_stAxis.stconfig.fReadAxisParameter := fbReadParameter.Value;
mParameters_ReadParameter.Busy := fbReadParameter.Busy;
mParameters_ReadParameter.Done := fbReadParameter.Valid;
mParameters_ReadParameter.Error := fbReadParameter.Error;
mParameters_ReadParameter.ErrorID := fbReadParameter.ErrorID;

IF fbReadParameter.Error THEN
    _stAxis.stError.fbReadParameterErrorId := fbReadParameter.ErrorID;
END_IF
END_METHOD

METHOD mParameters_WriteParameter : ST_McStatus

IF _stAxis.stControl.eCommand = E_MotionFunctions.eWriteParameter THEN
    fbWriteParameter.Execute := _stAxis.stControl.bExecute;
END_IF

fbWriteParameter.ParameterNumber := _stAxis.stConfig.eAxisParameters;
fbWriteParameter.Value := _stAxis.stConfig.fWriteAxisParameter;

fbWriteParameter(Axis := _stAxis.Axis);
fbWriteParameter.Execute := FALSE;

mParameters_WriteParameter.Busy := fbWriteParameter.Busy;
mParameters_WriteParameter.Done := fbWriteParameter.Done;
mParameters_WriteParameter.Error := fbWriteParameter.Error;
mParameters_WriteParameter.ErrorID := fbWriteParameter.ErrorID;

IF fbWriteParameter.Error THEN
    _stAxis.stError.fbWriteParameterErrorId := fbWriteParameter.ErrorID;
END_IF
END_METHOD

METHOD mParameters_WriteSWLimits : ST_McStatus
IF _stAxis.stControl.eCommand = E_MotionFunctions.eWriteToggleSWLimits THEN
    fbWriteSWLimitMax.Execute := _stAxis.stControl.bExecute;
	fbWriteSWLimitMin.Execute := _stAxis.stControl.bExecute;
END_IF

fbWriteSWLimitMax.ParameterNumber := E_AxisParameters.EnableLimitForward;
fbWriteSWLimitMax.Value := _stAxis.stConfig.fWriteAxisBoolParameter;
fbWriteSWLimitMin.ParameterNumber := E_AxisParameters.EnableLimitBackward;
fbWriteSWLimitMin.Value := _stAxis.stConfig.fWriteAxisBoolParameter;

fbWriteSWLimitMax(Axis := _stAxis.Axis);
fbWriteSWLimitMax.Execute := FALSE;
fbWriteSWLimitMin(Axis := _stAxis.Axis);
fbWriteSWLimitMin.Execute := FALSE;

mParameters_WriteSWLimits.Busy := fbWriteSWLimitMax.Busy OR fbWriteSWLimitMin.Busy;
mParameters_WriteSWLimits.Done := fbWriteSWLimitMax.Done OR fbWriteSWLimitMin.Done;
mParameters_WriteSWLimits.Error := fbWriteSWLimitMax.Error OR fbWriteSWLimitMin.Error;
mParameters_WriteSWLimits.ErrorID := fbWriteSWLimitMax.ErrorID OR fbWriteSWLimitMin.ErrorID;

IF fbWriteSWLimitMax.Error OR fbWriteSWLimitMin.Error THEN
    _stAxis.stError.fbWriteParameterErrorId := fbWriteSWLimitMax.ErrorID OR fbWriteSWLimitMin.ErrorID; 
END_IF
END_METHOD

METHOD mStatus_AxisStatus : BOOL

_stAxis.Axis.ReadStatus();
IF _stAxis.Axis.Status.OpMode.Modulo THEN
    _stAxis.stStatus.fActPosition := _stAxis.Axis.NcToPlc.ModuloActPos;
ELSE
    _stAxis.stStatus.fActPosition := _stAxis.Axis.NcToPlc.ActPos;
END_IF

_stAxis.stStatus.bHomed := _stAxis.Axis.Status.Homed;
_stAxis.stStatus.bMoving := _stAxis.Axis.Status.Moving;
_stAxis.stStatus.fActVelocity := _stAxis.Axis.NcToPlc.ActVelo;
_stAxis.stStatus.bMovingForward := _stAxis.Axis.Status.PositiveDirection;
_stAxis.stStatus.bMovingBackward := _stAxis.Axis.Status.NegativeDirection;
_stAxis.stStatus.bInTargetPosition := _stAxis.Axis.Status.InTargetPosition;
//_stAxis.stStatus.bEnabled := _stAxis.Axis.Status.Operational;
_stAxis.stStatus.bEnabled := NOT(_stAxis.Axis.Status.Disabled);	//This is crap but I don't know a better way

_stAxis.stStatus.SPGEnabled := _stAxis.Axis.Status.ExtSetPointGenEnabled;
END_METHOD

METHOD mStatus_Busy : BOOL
VAR
    i: UINT;
    tmpBusy: BOOL;
END_VAR

FOR i := 5 TO 10 DO
    tmpBusy := astMcStatus[i]^.Busy OR tmpBusy;
END_FOR
mStatus_Busy := tmpBusy;
END_METHOD

METHOD mStatus_CommandAborted : BOOL
VAR
    i: UINT;
    tmpCmdAborted: BOOL;
END_VAR

FOR i := 5 TO 9 DO
    tmpCmdAborted := astMcStatus[i]^.CommandAborted OR tmpCmdAborted;
END_FOR

fbCommandAbortedRTrig(CLK := tmpCmdAborted);
IF fbCommandAbortedRTrig.Q THEN
    _stAxis.stStatus.bCommandAborted := TRUE;
END_IF
END_METHOD

METHOD mStatus_Done : BOOL
VAR
    i: UINT;
    tmpDone: BOOL;
END_VAR

FOR i := 5 TO 10 DO
    tmpDone := astMcStatus[i]^.Done OR tmpDone;
END_FOR
//fbDoneRTrig(CLK:= mStatus_Done());
fbDoneRTrig(CLK := tmpDone);
IF fbDoneRTrig.Q THEN
    _stAxis.stStatus.bDone := TRUE;
END_IF
END_METHOD

METHOD mStatus_Error : BOOL
VAR
    i: UINT;
    tmpError: BOOL;

END_VAR

FOR i := 1 TO nMCSTATUS_ARRAY_SIZE DO
    tmpError := astMcStatus[i]^.Error OR tmpError;
END_FOR


fbErrorRTrig(CLK := tmpError);

//Check if NC is in error state and propogate
IF _stAxis.Axis.Status.ErrorStop OR _stAxis.Axis.Status.Error THEN
    _stAxis.stStatus.bError := _stAxis.Axis.Status.ErrorStop OR _stAxis.Axis.Status.Error;
    _stAxis.stStatus.nErrorID := _stAxis.Axis.Status.ErrorID;//NC Error ID
END_IF



IF fbErrorRTrig.Q THEN
        //For each mcStatus
        FOR i := 1 TO nMCSTATUS_ARRAY_SIZE DO
            //If there's an error present propagate
            IF astMcStatus[i]^.ErrorID <> 0 THEN
				_stAxis.stStatus.bMcError := TRUE;
                _stAxis.stStatus.nMcErrorID := astMcStatus[i]^.ErrorID;
            END_IF
        END_FOR
END_IF
END_METHOD

METHOD mStatus_InVelocity : BOOL
VAR
    i: UINT;
    tmpInVelocity: BOOL;
END_VAR
FOR i := 1 TO nMCSTATUS_ARRAY_SIZE DO
    tmpInVelocity := astMcStatus[i]^.InVelocity OR tmpInVelocity;
END_FOR
//fbInVelocityRTrig(CLK:= mStatus_InVelocity());
fbInVelocityRTrig(CLK := tmpInVelocity);
IF fbInVelocityRTrig.Q THEN
    _stAxis.stStatus.bInVelocity := TRUE;
END_IF

fbInVelocityFTrig(CLK := _stAxis.Axis.Status.ContinuousMotion);
IF fbInVelocityFTrig.Q THEN
    _stAxis.stStatus.bInVelocity := FALSE;
END_IF
END_METHOD

METHOD mStatus_Name : BOOL
VAR
	eAxisNames : E_AxisNames;
	sAxisName : STRING;
	sSpace : STRING := ' ';
END_VAR
eAxisNames := TO_INT(GVL.iAxis);
sAxisName := TO_STRING(eAxisNames);
FOR iNameCharacterIndex := 0 TO LEN(sAxisName) DO
	IF  F_ToCHR(sAxisName[iNameCharacterIndex]) = '_' THEN
		sAxisName[iNameCharacterIndex] := sSpace[0];
	END_IF
END_FOR
_stAxis.stDescription.sAxisName := sAxisName;
END_METHOD

METHOD mStatus_NewCommand : BOOL
VAR
    i: UINT;
END_VAR

fbExecuteRTrig(CLK := _stAxis.stControl.bExecute);
IF fbExecuteRTrig.Q THEN
    _stAxis.stStatus.bDone := FALSE;
    _stAxis.stStatus.bCommandAborted := FALSE;

    //On a new motion command, clear the errorID
    CASE _stAxis.stControl.eCommand OF
            E_MotionFunctions.eMoveAbsolute,
            E_MotionFunctions.eMoveRelative,
            E_MotionFunctions.eMoveVelocity,
            E_MotionFunctions.eMoveModulo,
			E_MotionFunctions.eSetPosition,
            E_MotionFunctions.eHome :
                _stAxis.stStatus.nErrorID := 0;
            E_MotionFunctions.eWriteParameter,
            E_MotionFunctions.eReadParameter :
            // Nothing
    END_CASE
END_IF
END_METHOD

METHOD Run : BOOL
mStatus_AxisStatus();
mParameters_ReadNc();
mParameters_Init();
stMcStatusReadParameter := mParameters_ReadParameter();
stMcStatusWriteParameter := mParameters_WriteParameter();
stMcStatusWriteSWLimits := mParameters_WriteSWLimits();

mControl_LimitHitTimer();
mControl_LimitLinking();
mControl_LimitEdge();
stMcStatusPower := mControl_Power();
mControl_AutoEnableDisable();

mControl_EnableSPG();
mControl_DisableSPG();
mControl_FeedSPG();

stMcStatusHalt := mMove_Halt();
stMcStatusStop := mMove_Stop();
stMcStatusReset := mControl_Reset();
stMcStatusSetPosition := mMove_SetPosition();

stMcStatusMoveAbsolute := mMove_MoveAbsolute();
stMcStatusMoveRelative := mMove_MoveRelative();
stMcStatusMoveModulo := mMove_MoveModulo();
stMcStatusMoveVelocity := mMove_MoveVelocity();

stMcStatusLocalMoveAbsolute := mLocalMove_MoveAbsolute();
stMcStatusLocalMoveRelative := mLocalMove_MoveRelative();
stMcStatusLocalMoveVelocity := mLocalMove_MoveVelocity();

stMcStatusHome := mControl_Home();

mStatus_NewCommand();
mStatus_Done();
mStatus_Error();
mStatus_InVelocity();
mStatus_CommandAborted();
_stAxis.stStatus.bBusy := mStatus_Busy();

IF _TaskInfo[fbGetCurTaskIndex.index].FirstCycle THEN
	mStatus_Name();
END_IF


EndOfCycle();
END_METHOD

PROPERTY stAxis : REFERENCE TO ST_AxisStruct
GET
stAxis REF= _stAxis;
END_GET
SET
_stAxis REF= stAxis;
END_SET
END_PROPERTY

END_FUNCTION_BLOCK

// ---- tc_mca_std_lib/POUs/Motion/Homing/FB_Homing.TcPOU
FUNCTION_BLOCK FB_Homing
VAR_IN_OUT
    AxisRef: AXIS_REF;
	
END_VAR
VAR_INPUT
    bExecute: BOOL;
    bLimitFwd: BOOL;
    bLimitBwd: BOOL;
    bHomeSensor: BOOL;
    eHomeSeq: E_HomingRoutines;
    fHomePosition: LREAL;
    fHomeFinishDistance: LREAL;
	fHomeAbsPosition : LREAL;
	bDoAbsoluteMove : BOOL;
	fHomeMidRelativeMove : LREAL;
    stConfig: ST_AxisConfig;
	stHomingConfig : ST_AxisHomingConfig;
	bGoToFwdLimitFirst : BOOL;
	bGoToBwdLimitFirst : BOOL;
	fFastVelocity : LREAL;
END_VAR
VAR_OUTPUT
    bDone : BOOL;
    bBusy: BOOL;
    bCommandAborted: BOOL;
    bError: BOOL;
    nErrorId: UDINT;
	bInHomingSequence: BOOL;
END_VAR
VAR
    //Beckhoff homing function blocks
    fbStepLimitSwitchPreparation: MC_StepLimitSwitchDetection;
    fbStepLimitSwitchDetection: MC_StepLimitSwitchDetection;
    fbStepAbsoluteSwitchDetection: MC_StepAbsoluteSwitchDetection;
	fbStepAbsoluteSwitchPreparation: MC_StepAbsoluteSwitchDetection;
	fbStepReferencePulsePreparation: MC_StepReferencePulseDetection;
    fbStepReferencePulseDetection: MC_StepReferencePulseDetection;
    fbStepBlockLagDetection: MC_StepBlockLagBasedDetection;
    fbHomeDirect: MC_HomeDirect;
    fbSetPos: MC_SetPosition;
    fbFinishHoming: MC_FinishHoming;
    fbAbortHoming: MC_AbortHoming;
	fbMoveRelative : MC_MoveRelative;
	fbMoveAbsolute : MC_MoveAbsolute;
	fbMoveVelocity : MC_MoveVelocity;
    //Hardware Signals
    eLimitSwitchMode: MC_Switch_Mode := mcRisingEdge;
    stLimitSwitchSignal: MC_Ref_Signal_Ref;
    eRefSwitchMode: MC_Switch_Mode := mcRisingEdge;
    stRefSwitchSignal: MC_Ref_Signal_Ref;
    stEncPulseSignal: MC_Ref_Signal_Ref;
    //Homing parameters
    stPreparationDirection: MC_Home_Direction;
    stDetectDirection: MC_Home_Direction;
    stHomingParameter: MC_HomingParameter;
    stOptions: ST_Home_Options4;
    stOptions3: ST_Home_Options3;
    fbVelocityToCam: MC_ReadParameter;
    fVelocityToCam: LREAL;
    fbVelocityFromCam: MC_ReadParameter;
    fVelocityFromCam: LREAL;
    //State machine
    fbExecute: R_TRIG;
    bViaLimitSwitch: BOOL;
	bViaFastEncPulse : BOOL;
	bViaFastRef : BOOL;
    eHomingState: (eWaitForRequest := 0, ePreparation := 1, eDetection := 2, eSetPos := 3, eFinishHoming := 4, eMoveRelative:=5, eAbsMove:=6, eAbortHoming := 20, eGoToFwd:=7, eGoToBwd:=8, eWaitForFwd:=9,eWaitForBwd:=10);
    iErrorId: UDINT;
    bDetectionFB_Execute: BOOL;
    bDetectionFB_Done: BOOL;
    bDetectionFB_Busy: BOOL;
    bDetectionFB_CommandAborted: BOOL;
    bDetectionFB_Error: BOOL;
    nDetectionFB_ErrorID: UDINT;
    fRecordedPosition: LREAL;
    fRecordedPositionLatched: LREAL;
END_VAR

bInHomingSequence:= FALSE;
//Hardware signals
stLimitSwitchSignal.SignalSource := SignalSource_Default;
stLimitSwitchSignal.TouchProbe := PlcEvent;
stRefSwitchSignal.SignalSource := SignalSource_Default;
stRefSwitchSignal.TouchProbe := PlcEvent;
stRefSwitchSignal.Level := bHomeSensor;
stEncPulseSignal.SignalSource := SignalSource_ZeroPulse;
stEncPulseSignal.TouchProbe := TouchProbe1;

fbMoveRelative(
	Axis:= AxisRef, Velocity:= fVelocityToCam);
	fbMoveRelative.Execute:= FALSE;

fbMoveAbsolute(
	Axis:= AxisRef, Velocity:= fFastVelocity, Position:= fHomeAbsPosition);
	fbMoveAbsolute.Execute:= FALSE;

//Constantly read the NC for homing velocities so they are available when a homing is executed
fbVelocityToCam(
    Axis := AxisRef,
    Enable := TRUE,
    ParameterNumber := E_AxisParameters.AxisVelocityToCam,
    ReadMode := READMODE_CYCLIC);

fbVelocityFromCam(
    Axis := AxisRef,
    Enable := TRUE,
    ParameterNumber := E_AxisParameters.AxisVelocityFromCam,
    ReadMode := READMODE_CYCLIC);

    //Only write velocity if the function block has not errored
IF NOT fbVelocityToCam.Error THEN
    fVelocityToCam := fbVelocityToCam.Value;
END_IF

IF NOT fbVelocityFromCam.Error THEN
    fVelocityFromCam := fbVelocityFromCam.Value;
END_IF

    //Feeds function block errors through
IF fbVelocityToCam.Error THEN
    bError := TRUE;
    nErrorID := fbVelocityToCam.ErrorID;

ELSIF fbVelocityFromCam.Error THEN
    bError := TRUE;
    nErrorID := fbVelocityFromCam.ErrorID;
END_IF

//Common function blocks used for all routines
stOptions.DisableDriveAccess := stHomingConfig.bDisableDriveAccess;

//For StepBlockLagDetection
stOptions3.DisableDriveAccess := stHomingConfig.bDisableDriveAccess;

fbStepLimitSwitchPreparation.Options.DisableDriveAccess := stOptions.DisableDriveAccess;
fbStepLimitSwitchPreparation(
    Axis := AxisRef,
    Parameter := stHomingParameter,
    Direction := stPreparationDirection,
    LimitSwitchMode:= eLimitSwitchMode,
    LimitSwitchSignal:= stLimitSwitchSignal,
    Velocity := fVelocityToCam);
	


fbSetPos(
    Axis := AxisRef,
    Position := AxisRef.NcToPlc.ActPos - fRecordedPositionLatched + fHomePosition);

fbFinishHoming.Options.DisableDriveAccess := stOptions.DisableDriveAccess;
fbFinishHoming(
    Axis := AxisRef,
    Parameter := stHomingParameter,
    Velocity := fVelocityFromCam);

fbMoveVelocity(Axis:= AxisRef, Velocity:= ABS(fFastVelocity));
	fbMoveVelocity.Execute:= FALSE;

fbAbortHoming.Options.DisableDriveAccess := stOptions.DisableDriveAccess;
fbAbortHoming(
    Axis := AxisRef,
    Parameter := stHomingParameter);

//ACTs contain function blocks custom to each individual routine for the detection stage
CASE eHomeSeq OF
    E_HomingRoutines.eHomeToLimit_Bwd,
    E_HomingRoutines.eHomeToLimit_Fwd:
        actHomeToLimit();

    E_HomingRoutines.eHomeToRef_Bwd,
	E_HomingRoutines.eHomeToRef_Bwd_Fast,
	E_HomingRoutines.eHomeToRef_Fwd_Fast,
    E_HomingRoutines.eHomeToRef_Fwd:
        actHomeToRef();

    E_HomingRoutines.eHomeToEncPulse_Bwd,
    E_HomingRoutines.eHomeToEncPulse_Fwd,
    E_HomingRoutines.eHomeToEncPulse_viaBwdLimit,
    E_HomingRoutines.eHomeToEncPulse_viaFwdLimit,
	E_HomingRoutines.eHomeToEncPulse_BWD_FAST,
	E_HomingRoutines.eHomeToEncPulse_FWD_FAST:
        actHomeToEncPulse();

    E_HomingRoutines.eHomeToBlock_Bwd,
    E_HomingRoutines.eHomeToBlock_Fwd:
        actHomeToBlock();

    E_HomingRoutines.eHomeDirect:
        actHomeDirect();
END_CASE


//State machine
fbExecute(CLK:= bExecute);
CASE eHomingState OF

    eWaitForRequest:
        IF NOT bExecute THEN
            bBusy := FALSE;
            bDone := FALSE;
            bCommandAborted := FALSE;
            bError := FALSE;
            nErrorID := 0;
            iErrorID := 0;

            fbStepLimitSwitchPreparation.Execute := FALSE;
            fbStepLimitSwitchDetection.Execute := FALSE;
            fbStepAbsoluteSwitchDetection.Execute := FALSE;
			fbStepReferencePulsePreparation.Execute := FALSE;
            fbStepReferencePulseDetection.Execute := FALSE;
            fbStepBlockLagDetection.Execute := FALSE;
            fbHomeDirect.Execute := FALSE;
            fbSetPos.Execute := FALSE;
            fbFinishHoming.Execute := FALSE;
            fbAbortHoming.Execute := FALSE;
        END_IF

        IF fbExecute.Q AND NOT(eHomeSeq = E_HomingRoutines.eNoHoming)THEN
            bBusy:= TRUE;
			IF bGoToFwdLimitFirst THEN
				eHomingState:= eGoToFwd;
			ELSIF bGoToBwdLimitFirst THEN
				eHomingState:= eGoToBwd;
			ELSE
				eHomingState:= ePreparation;
			END_IF            
        END_IF

	eGoToFwd:
		fbMoveVelocity.Execute:= TRUE;
		fbMoveVelocity.Direction:= MC_Direction.MC_Positive_Direction;
		eHomingState:= eWaitForFwd;
		bInHomingSequence:= TRUE;
		
	eWaitForFwd:
		IF NOT bLimitFwd THEN
			eHomingState:= ePreparation;
		END_IF
		bInHomingSequence:= TRUE;
		//IF NOT fbMoveVelocity.Active THEN
		//	eHomingState:= eAbortHoming;
		//END_IF
		
	eGoToBwd:
		fbMoveVelocity.Direction:= MC_Direction.MC_Negative_Direction;
		fbMoveVelocity.Execute:= TRUE;
		eHomingState:= eWaitForBwd;
		bInHomingSequence:= TRUE;
		
	eWaitForBwd:
		IF NOT bLimitBwd THEN
			eHomingState:= ePreparation;
		END_IF
		bInHomingSequence:= TRUE;
		//IF NOT fbMoveVelocity.Active THEN
		//	eHomingState:= eAbortHoming;
		//END_IF

    ePreparation: //If bViaLimitSwitch is set TRUE then go first to a limit otherwise skip this step
		bInHomingSequence:= TRUE;
        IF bViaLimitSwitch THEN
            fbStepLimitSwitchPreparation.Execute := TRUE;
        ELSIF bViaFastEncPulse THEN
			fbStepReferencePulsePreparation.Execute := TRUE;
		ELSIF bViaFastRef THEN
			fbStepAbsoluteSwitchPreparation.Execute:= TRUE;
		ELSE
            eHomingState := eDetection;
        END_IF

		IF bViaLimitSwitch THEN
        	IF NOT fbStepLimitSwitchPreparation.Busy AND fbStepLimitSwitchPreparation.Done THEN
            	fbStepLimitSwitchPreparation.Execute := FALSE;
            	eHomingState := eDetection;
        	ELSIF NOT fbStepLimitSwitchPreparation.Busy AND (fbStepLimitSwitchPreparation.Error OR fbStepLimitSwitchPreparation.CommandAborted) THEN
            	iErrorID := fbStepLimitSwitchPreparation.ErrorID;
            	fbStepLimitSwitchPreparation.Execute := FALSE;
            	eHomingState := eAbortHoming;
        	END_IF
		END_IF
		IF bViaFastEncPulse THEN
			IF NOT fbStepReferencePulsePreparation.Busy AND fbStepReferencePulsePreparation.Done THEN
            	fbStepReferencePulsePreparation.Execute := FALSE;
            	eHomingState := eMoveRelative;
        	ELSIF NOT fbStepReferencePulsePreparation.Busy AND (fbStepReferencePulsePreparation.Error OR fbStepReferencePulsePreparation.CommandAborted) THEN
            	iErrorID := fbStepReferencePulsePreparation.ErrorID;
            	fbStepReferencePulsePreparation.Execute := FALSE;
            	eHomingState := eAbortHoming;
        	END_IF			
		END_IF
		IF bViaFastRef THEN
			IF NOT fbStepAbsoluteSwitchPreparation.Busy AND fbStepAbsoluteSwitchPreparation.Done THEN
            	fbStepAbsoluteSwitchPreparation.Execute := FALSE;
            	eHomingState := eMoveRelative;
        	ELSIF NOT fbStepAbsoluteSwitchPreparation.Busy AND (fbStepAbsoluteSwitchPreparation.Error OR fbStepAbsoluteSwitchPreparation.CommandAborted) THEN
            	iErrorID := fbStepAbsoluteSwitchPreparation.ErrorID;
            	fbStepAbsoluteSwitchPreparation.Execute := FALSE;
            	eHomingState := eAbortHoming;
        	END_IF			
		END_IF
		
	eMoveRelative:
		bInHomingSequence:= TRUE;
		fbMoveRelative.Execute:= TRUE;
		IF NOT fbMoveRelative.Busy AND fbMoveRelative.Done THEN
            	fbMoveRelative.Execute := FALSE;
            	eHomingState := eDetection;
        	ELSIF NOT fbMoveRelative.Busy AND (fbMoveRelative.Error OR fbMoveRelative.CommandAborted) THEN
            	iErrorID := fbMoveRelative.ErrorID;
            	fbMoveRelative.Execute := FALSE;
            	eHomingState := eAbortHoming;
        	END_IF


    eDetection: //Use bDetectionFB_<BOOL Variables> to interact with different detection FBs located in ACTs
		bInHomingSequence:= FALSE;
        bDetectionFB_Execute := TRUE;

        IF NOT bDetectionFB_Busy AND bDetectionFB_Done THEN
            bDetectionFB_Execute := FALSE;
            fRecordedPositionLatched := fRecordedPosition;
            IF eHomeSeq = E_HomingRoutines.eHomeDirect THEN
                bBusy := fbHomeDirect.Busy;
                bDone := fbHomeDirect.Done;
                bCommandAborted := fbHomeDirect.CommandAborted;
                bError := fbHomeDirect.Error;
                nErrorId := fbHomeDirect.ErrorID;
                eHomingState := eWaitForRequest;
            ELSE
                eHomingState := eSetPos;
            END_IF
        ELSIF NOT bDetectionFB_Busy AND (bDetectionFB_Error OR bDetectionFB_CommandAborted) THEN
            iErrorID := nDetectionFB_ErrorID;
            bDetectionFB_Execute := FALSE;
            eHomingState := eAbortHoming;
        END_IF


    eSetPos:
		bInHomingSequence:= FALSE;
        fbSetPos.Execute := TRUE;

        fbSetPos.Options.ClearPositionLag := TRUE;
        IF NOT fbSetPos.Busy AND fbSetPos.Done THEN
            fbSetPos.Execute := FALSE;
			IF bDoAbsoluteMove THEN
				eHomingState := eAbsMove;
			ELSE
				 eHomingState := eFinishHoming;
			END_IF
			
           
        ELSIF NOT fbSetPos.Busy AND fbSetPos.Error THEN
            iErrorID := fbSetPos.ErrorID;
            fbSetPos.Execute := FALSE;
            eHomingState := eAbortHoming;
        END_IF
	
	eAbsMove:
		bInHomingSequence:= FALSE;
		fbMoveAbsolute.Execute:= TRUE;
		IF NOT fbMoveAbsolute.Busy AND fbMoveAbsolute.Done THEN
            fbMoveAbsolute.Execute := FALSE;
            eHomingState := eFinishHoming;
        ELSIF NOT fbMoveAbsolute.Busy AND (fbMoveAbsolute.Error OR fbMoveAbsolute.CommandAborted) THEN
            iErrorID := fbMoveAbsolute.ErrorID;
            fbMoveAbsolute.Execute := FALSE;
            eHomingState := eAbortHoming;
        END_IF

    eFinishHoming:
		bInHomingSequence:= FALSE;
        fbFinishHoming.Execute := TRUE;

        IF NOT fbFinishHoming.Busy AND fbFinishHoming.Done THEN
            bBusy := FALSE;
            bDone := TRUE;
            fbFinishHoming.Execute := FALSE;
            eHomingState := eWaitForRequest;
        ELSIF NOT fbFinishHoming.Busy AND (fbFinishHoming.Error OR fbFinishHoming.CommandAborted) THEN
            iErrorID := fbFinishHoming.ErrorID;
            fbFinishHoming.Execute := FALSE;
            eHomingState := eAbortHoming;
        END_IF


    eAbortHoming:
		bInHomingSequence:= FALSE;
        fbAbortHoming.Execute := TRUE;

        IF NOT fbAbortHoming.Busy AND fbAbortHoming.Done THEN
            bBusy := FALSE;
            IF iErrorId <> 0 THEN
                bError := TRUE;
                nErrorId := iErrorId;
            ELSE
                bCommandAborted := TRUE;
            END_IF
            fbAbortHoming.Execute := FALSE;
            eHomingState := eWaitForRequest;
        ELSIF NOT fbAbortHoming.Busy AND fbAbortHoming.Error THEN
            bBusy := FALSE;
            bError := TRUE;
            nErrorID := fbAbortHoming.ErrorID;
            fbAbortHoming.Execute := FALSE;
            eHomingState := eWaitForRequest;
        END_IF

END_CASE

ACTION actHomeDirect:

bViaLimitSwitch := FALSE;

fbHomeDirect(
    Axis := AxisRef,
    Parameter := stHomingParameter,
    Execute := bDetectionFB_Execute,
    SetPosition := fHomePosition,
    Done => bDetectionFB_Done,
    Busy => bDetectionFB_Busy,
    CommandAborted => bDetectionFB_CommandAborted,
    Error => bDetectionFB_Error,
    ErrorID => nDetectionFB_ErrorID);
END_ACTION

ACTION actHomeToBlock:
CASE eHomeSeq OF
    E_HomingRoutines.eHomeToBlock_Bwd:
        stDetectDirection:= mcNegativeDirection;
        fbFinishHoming.Distance := fHomeFinishDistance;
    E_HomingRoutines.eHomeToBlock_Fwd:
        stDetectDirection:= mcPositiveDirection;
        fbFinishHoming.Distance := -fHomeFinishDistance;
END_CASE

bViaLimitSwitch:=FALSE;

fbStepBlockLagDetection(
    Axis := AxisRef,
    Execute := bDetectionFB_Execute,
    Parameter := stHomingParameter,
    Direction := stDetectDirection,
    Velocity := fVelocityFromCam, //Maximum travel velocity (>0).
    DetectionVelocityLimit := stHomingConfig.fDetectionVelocityLimit, //Velocity that must be fallen below for the time DetectionVelocityTime in order to detect driving against the fixed stop.
    DetectionVelocityTime := stHomingConfig.tDetectionVelocityTime, //Time for detecting the velocity undershoot when driving against the fixed stop.
    TimeLimit :=  stHomingConfig.tTimeLimit, //Exceeding this time leads to the search procedure being aborted.
    DistanceLimit := stHomingConfig.fDistanceLimit, //Exceeding this distance in relation to the start position leads to the search procedure being aborted.
    TorqueLimit := stHomingConfig.fTorqueLimit, //The motor torque is limited to this value (percentage of configured channel peak torque), in relation to the weight counterbalance that is possibly parameterized in the drive, in order to avoid mechanical damage.
    LagLimit := stHomingConfig.fLagLimit, //Position lag value which, if exceeded, leads to detection of driving against the fixed stop.
    Options := stOptions3,
    Done => bDetectionFB_Done,
    Busy => bDetectionFB_Busy,
    CommandAborted => bDetectionFB_CommandAborted,
    Error => bDetectionFB_Error,
    ErrorID => nDetectionFB_ErrorID,
    RecordedPosition => fRecordedPosition);
END_ACTION

ACTION actHomeToEncPulse:

CASE eHomeSeq OF
    E_HomingRoutines.eHomeToEncPulse_Bwd:
        stDetectDirection := mcNegativeDirection;
        fbFinishHoming.Distance := fHomeFinishDistance;
        bViaLimitSwitch := FALSE;
		bViaFastEncPulse:= FALSE;
		bViaFastRef := FALSE;
    E_HomingRoutines.eHomeToEncPulse_Fwd:
        stDetectDirection := mcPositiveDirection;
        fbFinishHoming.Distance := -fHomeFinishDistance;
        bViaLimitSwitch := FALSE;
		bViaFastEncPulse:= FALSE;
		bViaFastRef := FALSE;
    E_HomingRoutines.eHomeToEncPulse_viaBwdLimit:
        stDetectDirection := mcPositiveDirection;
        fbFinishHoming.Distance := fHomeFinishDistance;
        stPreparationDirection := mcNegativeDirection;
        stLimitSwitchSignal.Level := NOT(bLimitBwd);
        bViaLimitSwitch := TRUE;
		bViaFastEncPulse:= FALSE;
		bViaFastRef := FALSE;
    E_HomingRoutines.eHomeToEncPulse_viaFwdLimit:
        stDetectDirection := mcNegativeDirection;
        fbFinishHoming.Distance := -fHomeFinishDistance;
        stPreparationDirection := mcPositiveDirection;
        stLimitSwitchSignal.Level := NOT(bLimitFwd);
        bViaLimitSwitch := TRUE;
		bViaFastEncPulse:= FALSE;
		bViaFastRef := FALSE;
	
	E_HomingRoutines.eHomeToEncPulse_BWD_FAST:
		stDetectDirection := mcNegativeDirection;
        fbFinishHoming.Distance := fHomeFinishDistance;
        bViaLimitSwitch := FALSE;
		bViaFastEncPulse:= TRUE;
		bViaFastRef := FALSE;
		fbMoveRelative.Distance:= ABS(fHomeMidRelativeMove);
	
	E_HomingRoutines.eHomeToEncPulse_FWD_FAST:
		stDetectDirection := mcPositiveDirection;
        fbFinishHoming.Distance := fHomeFinishDistance;
        bViaLimitSwitch := FALSE;
		bViaFastEncPulse:= TRUE;
		fbMoveRelative.Distance:= -ABS(fHomeMidRelativeMove);
END_CASE

fbStepReferencePulsePreparation.Options.DisableDriveAccess := stOptions.DisableDriveAccess;
fbStepReferencePulsePreparation(
    Axis := AxisRef,
    Parameter := stHomingParameter,
    Direction := stDetectDirection,
    ReferenceSignal := stEncPulseSignal,
    Velocity := fVelocityToCam,
    Options := stOptions);
	

fbStepReferencePulseDetection.Options.DisableDriveAccess:= stOptions.DisableDriveAccess;
fbStepReferencePulseDetection(
    Axis := AxisRef,
    Execute := bDetectionFB_Execute,
    Parameter := stHomingParameter,
    Direction := stDetectDirection,
    ReferenceSignal := stEncPulseSignal,
    Velocity := fVelocityFromCam,
    Options := stOptions,
    Done => bDetectionFB_Done,
    Busy => bDetectionFB_Busy,
    CommandAborted => bDetectionFB_CommandAborted,
    Error => bDetectionFB_Error,
    ErrorID => nDetectionFB_ErrorID,
    RecordedPosition => fRecordedPosition);
END_ACTION

ACTION actHomeToLimit:

CASE eHomeSeq OF
    E_HomingRoutines.eHomeToLimit_Bwd:
        stLimitSwitchSignal.Level := NOT(bLimitBwd);
        stDetectDirection:= mcNegativeDirection;
        fbFinishHoming.Distance := fHomeFinishDistance;
    E_HomingRoutines.eHomeToLimit_Fwd:
        stLimitSwitchSignal.Level := NOT(bLimitFwd);
        stDetectDirection:= mcPositiveDirection;
        fbFinishHoming.Distance := -fHomeFinishDistance;
END_CASE
bViaLimitSwitch:=FALSE;

fbStepLimitSwitchDetection.Options.DisableDriveAccess:= stOptions.DisableDriveAccess;
fbStepLimitSwitchDetection(
    Axis := AxisRef,
    Execute := bDetectionFB_Execute,
    Parameter := stHomingParameter,
    Direction := stDetectDirection,
    LimitSwitchMode := eLimitSwitchMode,
    LimitSwitchSignal := stLimitSwitchSignal,
    Velocity := fVelocityFromCam,
    Options := stOptions,
    Done => bDetectionFB_Done,
    Busy => bDetectionFB_Busy,
    CommandAborted => bDetectionFB_CommandAborted,
    Error => bDetectionFB_Error,
    ErrorID => nDetectionFB_ErrorID,
    RecordedPosition => fRecordedPosition);
END_ACTION

ACTION actHomeToRef:

CASE eHomeSeq OF
    E_HomingRoutines.eHomeToRef_Bwd:
        stDetectDirection := mcNegativeDirection;
        fbFinishHoming.Distance := fHomeFinishDistance;
		bViaFastRef := FALSE;
		bViaLimitSwitch := FALSE;
		bViaFastEncPulse:= FALSE;
		
    E_HomingRoutines.eHomeToRef_Fwd:
        stDetectDirection := mcPositiveDirection;
        fbFinishHoming.Distance := -fHomeFinishDistance;
		bViaFastRef := FALSE;
		bViaLimitSwitch := FALSE;
		bViaFastEncPulse:= FALSE;
		
	E_HomingRoutines.eHomeToRef_Bwd_Fast:
        stDetectDirection := mcNegativeDirection;
        fbFinishHoming.Distance := fHomeFinishDistance;
		fbMoveRelative.Distance:= ABS(fHomeMidRelativeMove);
		bViaFastRef := TRUE;
		bViaLimitSwitch := FALSE;
		bViaFastEncPulse:= FALSE;
		
    E_HomingRoutines.eHomeToRef_Fwd_Fast:
        stDetectDirection := mcPositiveDirection;
        fbFinishHoming.Distance := -fHomeFinishDistance;
		fbMoveRelative.Distance:= -ABS(fHomeMidRelativeMove);
		bViaFastRef := TRUE;
		bViaLimitSwitch := FALSE;
		bViaFastEncPulse:= FALSE;
		
END_CASE
bViaLimitSwitch := FALSE;

fbStepAbsoluteSwitchDetection.Options.DisableDriveAccess := stOptions.DisableDriveAccess;
fbStepAbsoluteSwitchDetection(
    Axis := AxisRef,
    Execute := bDetectionFB_Execute,
    Parameter := stHomingParameter,
    Direction := stDetectDirection,
    SwitchMode := eRefSwitchMode,
    ReferenceSignal := stRefSwitchSignal,
    Velocity := fVelocityFromCam,
    PositiveLimitSwitch := NOT(bLimitFwd),
    NegativeLimitSwitch := NOT(bLimitBwd),
    Options := stOptions,
    Done => bDetectionFB_Done,
    Busy => bDetectionFB_Busy,
    CommandAborted => bDetectionFB_CommandAborted,
    Error => bDetectionFB_Error,
    ErrorID => nDetectionFB_ErrorID,
    RecordedPosition => fRecordedPosition);
	
fbStepAbsoluteSwitchPreparation.Options.DisableDriveAccess := stOptions.DisableDriveAccess;
fbStepAbsoluteSwitchPreparation(
    Axis := AxisRef,
    Parameter := stHomingParameter,
    Direction := stDetectDirection,
    SwitchMode := eRefSwitchMode,
    ReferenceSignal := stRefSwitchSignal,
    Velocity := fVelocityToCam,
    PositiveLimitSwitch := NOT(bLimitFwd),
    NegativeLimitSwitch := NOT(bLimitBwd),
    Options := stOptions);
END_ACTION

END_FUNCTION_BLOCK

// ---- tc_mca_std_lib/POUs/Pneumatics/FB_PneumaticAxis.TcPOU

FUNCTION_BLOCK FB_PneumaticAxis

VAR_IN_OUT
    stPneumaticAxisStruct: ST_PneumaticAxisStruct;
END_VAR
VAR
    fbTimerExtend: TON; //Timing the extraction of the cylinder
    fbTimerRetract: TON; //Timing the retraction of the cylinder
    fbTrigRisingEdgePermit: R_TRIG; //Rising edge detection for Permit signal
    fbTrigExtendManual: R_TRIG; //Rising edge detection for manual push button
    fbTrigRetractManual: R_TRIG; //Rising edge detection for manual push button
    bStateChange: BOOL := FALSE; //State of the cylinder changed from extend to retract and vice versa
    bStartExtendManual: BOOL; //Variable to control the solenoid valve with momentary push button
    bStartRetractManual: BOOL; //VAriable to control the solenoid valve with momentary push button
END_VAR


Initialization();

CASE stPneumaticAxisStruct.ePneumaticAxisMode OF

    E_PneumaticMode.eSingleSolenoidControl:
    Single_Solenoid();

    E_PneumaticMode.eError:
    Single_Solenoid_Error();

    E_PneumaticMode.eReset:
    Reset();
END_CASE

ACTION ErrorCheck:
//IF the command to extract is given, but the cylinder hasn't moved from the bEndSwitchBwd
    IF  fbTimerExtend.Q AND stPneumaticAxisStruct.stPneumaticAxisStatus.bRetracted THEN
             stPneumaticAxisStruct.stPneumaticAxisStatus.bExtending := FALSE;
             stPneumaticAxisStruct.ePneumaticAxisMode := E_PneumaticMode.eError;
    END_IF
//If the command to extract has timed out
    IF  fbTimerExtend.Q AND (NOT stPneumaticAxisStruct.stPneumaticAxisStatus.bRetracted AND NOT stPneumaticAxisStruct.stPneumaticAxisStatus.bExtended) THEN
            stPneumaticAxisStruct.stPneumaticAxisStatus.bExtending := FALSE;
            stPneumaticAxisStruct.ePneumaticAxisMode := E_PneumaticMode.eError;
    END_IF

//IF the command to retract has been given, but the cylinder hasn't moved from bEndSwitchFwd
        IF  fbTimerRetract.Q AND stPneumaticAxisStruct.stPneumaticAxisStatus.bExtended THEN
            stPneumaticAxisStruct.stPneumaticAxisStatus.bRetracting := FALSE;
            stPneumaticAxisStruct.ePneumaticAxisMode := E_PneumaticMode.eError;
        END_IF

//If the command to retract has timed out
        IF  fbTimerRetract.Q AND (NOT stPneumaticAxisStruct.stPneumaticAxisStatus.bExtended AND NOT stPneumaticAxisStruct.stPneumaticAxisStatus.bRetracted) THEN
            stPneumaticAxisStruct.stPneumaticAxisStatus.bRetracting := FALSE;
            stPneumaticAxisStruct.ePneumaticAxisMode := E_PneumaticMode.eError;
        END_IF
END_ACTION

ACTION Initialization:
//Set the inputs of limit switches to bExtracted and bRetracted states of the pneumatic cylinders
stPneumaticAxisStruct.stPneumaticAxisStatus.bRetracted := stPneumaticAxisStruct.stPneumaticAxisInputs.bEndSwitchBwd;
stPneumaticAxisStruct.stPneumaticAxisStatus.bExtended := stPneumaticAxisStruct.stPneumaticAxisInputs.bEndSwitchFwd;
stPneumaticAxisStruct.stPneumaticAxisStatus.bSolenoidActive := stPneumaticAxisStruct.stPneumaticAxisInputs.bSolenoidActive;
stPneumaticAxisStruct.stPneumaticAxisStatus.bPSSPermitOK := stPneumaticAxisStruct.stPneumaticAxisInputs.bPSSPermit;
stPneumaticAxisStruct.stPneumaticAxisStatus.bInterlocked := stPneumaticAxisStruct.stPneumaticAxisControl.bInterlock;


//Check if Permit signal is ON
IF NOT stPneumaticAxisStruct.stPneumaticAxisInputs.bPSSPermit THEN
            stPneumaticAxisStruct.stPneumaticAxisOutputs.bValveOn := FALSE;
            stPneumaticAxisStruct.ePneumaticAxisMode := E_PneumaticMode.eError;
END_IF

//Reset Error
fbTrigRisingEdgePermit(clk:=stPneumaticAxisStruct.stPneumaticAxisControl.bReset);

IF fbTrigRisingEdgePermit.Q THEN
    stPneumaticAxisStruct.ePneumaticAxisMode := E_PneumaticMode.eReset;
END_IF

//Check if Interlock signal is ON
IF stPneumaticAxisStruct.stPneumaticAxisControl.bInterlock THEN
            stPneumaticAxisStruct.stPneumaticAxisOutputs.bValveOn := FALSE;
            stPneumaticAxisStruct.ePneumaticAxisMode := E_PneumaticMode.eError;
END_IF

//Check for errors in Air pressure (to be implemented)
END_ACTION

ACTION Reset:
//Reset all the error messages
//Set the operating mode to Single Solenoid Control

stPneumaticAxisStruct.stPneumaticAxisStatus.sStatus := 'NO_ERRORS_READY_TO_START';
stPneumaticAxisStruct.ePneumaticAxisErrors := E_PneumaticAxisErrors.eNoError;
stPneumaticAxisStruct.stPneumaticAxisStatus.bError := FALSE;
stPneumaticAxisStruct.ePneumaticAxisMode := E_PneumaticMode.eSingleSolenoidControl;
END_ACTION

ACTION Single_Solenoid:
//Enter allowed times for extraction and retraction of pneumatic cylinder in seconds
 fbTimerExtend.PT := INT_TO_TIME( stPneumaticAxisStruct.stPneumaticAxisConfig.nTimeToExtend)*1000;
 fbTimerRetract.PT := INT_TO_TIME( stPneumaticAxisStruct.stPneumaticAxisConfig.nTimeToRetract)*1000;


//Starting the timing of extraction movement
fbTimerExtend();
fbTimerExtend(IN := stPneumaticAxisStruct.stPneumaticAxisStatus.bExtending);

//If the manual momentary push button is used for control of the pneumatic cylinder
fbTrigExtendManual(clk:=stPneumaticAxisStruct.stPneumaticAxisInputs.bOpenManual);

IF fbTrigExtendManual.Q THEN
    bStartExtendManual := TRUE;
END_IF

//Starting the extraction movement
IF (stPneumaticAxisStruct.stPneumaticAxisControl.bExtend OR bStartExtendManual) THEN
        stPneumaticAxisStruct.stPneumaticAxisOutputs.bValveOn := TRUE;
        stPneumaticAxisStruct.stPneumaticAxisStatus.bExtending := TRUE;
//If the command to retract is given while the cylinder is extracting
    IF NOT stPneumaticAxisStruct.stPneumaticAxisStatus.bExtended AND NOT stPneumaticAxisStruct.stPneumaticAxisStatus.bRetracted THEN
        IF (stPneumaticAxisStruct.stPneumaticAxisControl.bRetract OR bStartRetractManual) THEN
            stPneumaticAxisStruct.stPneumaticAxisOutputs.bValveOn := FALSE;
            stPneumaticAxisStruct.stPneumaticAxisStatus.bRetracting := TRUE;
            stPneumaticAxisStruct.stPneumaticAxisStatus.bExtending := FALSE;
            stPneumaticAxisStruct.stPneumaticAxisControl.bExtend := FALSE;
        bStartExtendManual := FALSE;
        END_IF
    END_IF


END_IF
//Check for errors while the cylinder is extending
ErrorCheck();

// Extraction of the cylinder finished, reset timer
IF (stPneumaticAxisStruct.stPneumaticAxisControl.bExtend OR bStartExtendManual) AND stPneumaticAxisStruct.stPneumaticAxisStatus.bExtended THEN
        bStateChange := TRUE;
        stPneumaticAxisStruct.stPneumaticAxisStatus.bExtending := FALSE;
        stPneumaticAxisStruct.stPneumaticAxisControl.bExtend := FALSE;
        bStartExtendManual := FALSE;
END_IF



//Starting the retraction movement and retraction timing
fbTimerRetract();
fbTimerRetract (IN := stPneumaticAxisStruct.stPneumaticAxisStatus.bRetracting);

//If the manual momentary push button is used for control of the pneumatic cylinder
fbTrigRetractManual(clk:=stPneumaticAxisStruct.stPneumaticAxisInputs.bCloseManual);

IF fbTrigRetractManual.Q THEN
    bStartRetractManual := TRUE;
END_IF

IF (stPneumaticAxisStruct.stPneumaticAxisControl.bRetract OR bStartRetractManual) THEN
        stPneumaticAxisStruct.stPneumaticAxisOutputs.bValveOn := FALSE;
        stPneumaticAxisStruct.stPneumaticAxisStatus.bRetracting := TRUE;


END_IF
//Check for errors while the cylinder is retracting
ErrorCheck();
// Retraction of the cylinder finished, reset timer
IF  (stPneumaticAxisStruct.stPneumaticAxisControl.bRetract OR bStartRetractManual) AND stPneumaticAxisStruct.stPneumaticAxisStatus.bRetracted THEN
        bStateChange := FALSE;
        stPneumaticAxisStruct.stPneumaticAxisStatus.bRetracting := FALSE;
        stPneumaticAxisStruct.stPneumaticAxisControl.bRetract := FALSE;
        bStartRetractManual := FALSE;
END_IF
END_ACTION

ACTION Single_Solenoid_Error:
IF NOT stPneumaticAxisStruct.stPneumaticAxisInputs.bPSSPermit THEN
    stPneumaticAxisStruct.ePneumaticAxisErrors := E_PneumaticAxisErrors.eNoPSSPermit;
END_IF

IF stPneumaticAxisStruct.stPneumaticAxisControl.bInterlock THEN
     stPneumaticAxisStruct.ePneumaticAxisErrors := E_PneumaticAxisErrors.eInterlockOn;
END_IF

IF  fbTimerExtend.Q AND stPneumaticAxisStruct.stPneumaticAxisStatus.bRetracted THEN
    stPneumaticAxisStruct.ePneumaticAxisErrors := E_PneumaticAxisErrors.eNotMovingExtract;
END_IF

IF  fbTimerExtend.Q AND NOT stPneumaticAxisStruct.stPneumaticAxisStatus.bRetracted AND NOT stPneumaticAxisStruct.stPneumaticAxisStatus.bExtended THEN
    stPneumaticAxisStruct.ePneumaticAxisErrors := E_PneumaticAxisErrors.eExtractTimedOut;
END_IF

IF  fbTimerRetract.Q AND stPneumaticAxisStruct.stPneumaticAxisStatus.bExtended THEN
    stPneumaticAxisStruct.ePneumaticAxisErrors := E_PneumaticAxisErrors.eNotMovingRetract;
END_IF

IF  fbTimerRetract.Q AND NOT stPneumaticAxisStruct.stPneumaticAxisStatus.bExtended AND NOT stPneumaticAxisStruct.stPneumaticAxisStatus.bRetracted THEN
    stPneumaticAxisStruct.ePneumaticAxisErrors := E_PneumaticAxisErrors.eRetractTimedOut;
END_IF


CASE  stPneumaticAxisStruct.ePneumaticAxisErrors OF

    E_PneumaticAxisErrors.eNoError:
    stPneumaticAxisStruct.stPneumaticAxisStatus.bError := FALSE;

    E_PneumaticAxisErrors.eExtractTimedOut:
    stPneumaticAxisStruct.stPneumaticAxisStatus.sStatus := 'ERROR: COMMAND TIMED OUT';
    stPneumaticAxisStruct.stPneumaticAxisStatus.bError := TRUE;

    E_PneumaticAxisErrors.eRetractTimedOut:
    stPneumaticAxisStruct.stPneumaticAxisStatus.sStatus := 'ERROR: COMMAND TIMED OUT';
    stPneumaticAxisStruct.stPneumaticAxisStatus.bError := TRUE;

    E_PneumaticAxisErrors.eNotMovingExtract:
    stPneumaticAxisStruct.stPneumaticAxisStatus.sStatus := 'ERROR: CYLINDER NOT MOVING';
    stPneumaticAxisStruct.stPneumaticAxisStatus.bError := TRUE;

    E_PneumaticAxisErrors.eNotMovingRetract:
    stPneumaticAxisStruct.stPneumaticAxisStatus.sStatus := 'ERROR: CYLINDER NOT MOVING';
    stPneumaticAxisStruct.stPneumaticAxisStatus.bError := TRUE;

    E_PneumaticAxisErrors.eNoPSSPermit:
    stPneumaticAxisStruct.stPneumaticAxisStatus.sStatus := 'ERROR: NO PERMIT SIGNAL';
    stPneumaticAxisStruct.stPneumaticAxisStatus.bError := TRUE;

    E_PneumaticAxisErrors.eInterlockOn:
    stPneumaticAxisStruct.stPneumaticAxisStatus.sStatus := 'ERROR: INTERLOCK SIGNAL ON';
    stPneumaticAxisStruct.stPneumaticAxisStatus.bError := TRUE;

END_CASE

stPneumaticAxisStruct.stPneumaticAxisControl.bExtend := FALSE;
stPneumaticAxisStruct.stPneumaticAxisControl.bRetract := FALSE;
stPneumaticAxisStruct.stPneumaticAxisOutputs.bValveOn := FALSE;
bStartExtendManual := FALSE;
bStartRetractManual := FALSE;
stPneumaticAxisStruct.stPneumaticAxisStatus.bExtending := FALSE;
stPneumaticAxisStruct.stPneumaticAxisStatus.bRetracting := FALSE;
END_ACTION

END_FUNCTION_BLOCK

// ---- POUs/Application_Specific/Axes/Axis1.TcPOU
PROGRAM Axis1
VAR
	iAxisNumber : INT := E_AxisNames.Axis1;
	iGroupNumber : INT := 1;
	
	stoRTrig : R_Trig;
	
	//Automatic reset on permit
	startReset : BOOL;
	resetDelay : TON;
	startDisable : BOOL;
	disableDelay : TON;
END_VAR

//Initial parameters of an Axis

IF _TaskInfo[fbGetCurTaskIndex.index].FirstCycle THEN
    //Initial default values:
    GVL.astAxes[iAxisNumber].stHomingConfig.eHomeSeq :=E_HomingRoutines.eHomeToEncPulse_viaBwdLimit;
	GVL.astAxes[iAxisNumber].stHomingConfig.fHomeAbsPosition:= 0;
	GVL.astAxes[iAxisNumber].stHomingConfig.fHomeMidRelativeMove:=1;
    GVL.astAxes[iAxisNumber].stHomingConfig.fHomePosition := 0;
    GVL.astAxes[iAxisNumber].stHomingConfig.fHomeFinishDistance := 0.0;
    GVL.astAxes[iAxisNumber].stConfig.eRestorePosition := E_RestorePosition.eRestoreWithoutHome;
	GVL.astAxes[iAxisNumber].stControl.bAutoEnableDisable := TRUE;
	GVL.astAxes[iAxisNumber].stControl.tMoveFinishedDelay := T#0.1S;
	//Set which group this axis belongs to
	GVL.astAxes[iAxisNumber].stDescription.iGroupNumber := iGroupNumber;
	GVL.astAxes[iAxisNumber].Commissioning := FALSE;
	GVL.astAxes[iAxisNumber].stDescription.sUnits:= 'mm';
END_IF

//Permit
GVL.astAxes[iAxisNumber].stInputs.bPermit := TRUE;//(SAFETY.SAMPLE_PERMIT AND NOT SAFETY.CollisionDetected) OR (SAFETY.SAMPLE_PERMIT AND (safety.inMode_Local OR safety.inMode_Maintenance));

//Remote operation toggle

IF SAFETY.inMode_Local THEN
	GVL.astAxes[iAxisNumber].stInputs.bAllowRemoteControl:= FALSE;
ELSIF SAFETY.inMode_Maintenance AND NOT SAFETY.maintenanceAllowRemote THEN
	GVL.astAxes[iAxisNumber].stInputs.bAllowRemoteControl:= FALSE;
ELSE
	GVL.astAxes[iAxisNumber].stInputs.bAllowRemoteControl:= TRUE;
END_IF

//Do an automatic reset on regaining permit;

IF SAFETY.SAMPLE_PERMIT_R_EDGE THEN
	startReset:= TRUE;
END_IF
resetDelay(IN:= startReset, PT:= T#0.5S);
IF resetDelay.Q THEN
	startReset := FALSE;
	GVL.astAxes[iAxisNumber].stControl.bReset:= TRUE;
END_IF


//Disable axis if no permit

IF SAFETY.STOP_MOTION THEN
	startDisable := TRUE;
END_IF
disableDelay(IN:= startDisable, PT:= T#1S);
IF disableDelay.Q THEN
	startDisable:= FALSE;
	GVL.astAxes[iAxisNumber].stControl.bEnable:= FALSE;
END_IF



//Safety stop motion

IF SAFETY.STOP_MOTION THEN
	GVL.astAxes[iAxisNumber].stControl.bHalt:= TRUE;
END_IF
IF SAFETY.collisionDetected_R_Edge THEN
	GVL.astAxes[iAxisNumber].stControl.bHalt:= TRUE;
END_IF

stoRTrig(CLK:=GVL.astAxes[iAxisNumber].stStatus.bSTOActive);
IF stoRTrig.Q THEN
	GVL.astAxes[iAxisNumber].stControl.bReset:= TRUE;
END_IF

END_PROGRAM

// ---- POUs/SAFETY.TcPOU
PROGRAM SAFETY
VAR
SafetyTargets : ARRAY [1..7] OF ST_SafetyTargetDevice:=
[
//(ProjectName:='MAIN', Device:='EL6910',aSafetyGroups:=[(Connected:=TRUE),(Connected:=TRUE),(Connected:=TRUE),(Connected:=TRUE),(Connected:=TRUE),(Connected:=TRUE),(Connected:=TRUE),(Connected:=TRUE)]),
(ProjectName:='SampleStackZ', Device:='AX891x',aSafetyGroups:=[(Connected:=TRUE),(Connected:=TRUE),(Connected:=TRUE)]),
(ProjectName:='SampleStackRotation', Device:='AX891x',aSafetyGroups:=[(Connected:=TRUE),(Connected:=TRUE),(Connected:=TRUE),(Connected:=TRUE)]),
(ProjectName:='CollimationNorthX', Device:='AMI891x',aSafetyGroups:=[(Connected:=TRUE),(Connected:=TRUE),(Connected:=TRUE)]),
(ProjectName:='CollimationNorthY', Device:='AMI891x',aSafetyGroups:=[(Connected:=TRUE),(Connected:=TRUE),(Connected:=TRUE)]),
(ProjectName:='CollimationSouthX', Device:='AMI891x',aSafetyGroups:=[(Connected:=TRUE),(Connected:=TRUE),(Connected:=TRUE)]),
(ProjectName:='CollimationSouthY', Device:='AMI891x',aSafetyGroups:=[(Connected:=TRUE),(Connected:=TRUE),(Connected:=TRUE)])
]
;
	i : INT;
	j : INT;
	iGroup : INT;
	
	RUN AT %Q* : BOOL := TRUE;
	ERRACK AT %Q* : BOOL;
	
	BannerMessage : STRING;
	
	//ESTOP Devices
	{ attribute 'TcHmiSymbol.AddSymbol' }
	MS1 : ST_DeviceDualChannelInput;
	{ attribute 'TcHmiSymbol.AddSymbol' }
	MS2 : ST_DeviceDualChannelInput;
	{ attribute 'TcHmiSymbol.AddSymbol' }
	MS3 : ST_DeviceDualChannelInput;
	{ attribute 'TcHmiSymbol.AddSymbol' }
	MS4 : ST_DeviceDualChannelInput;
	{ attribute 'TcHmiSymbol.AddSymbol' }
	MS5 : ST_DeviceDualChannelInput;
	{ attribute 'TcHmiSymbol.AddSymbol' }
	MS6 : ST_DeviceDualChannelInput;
	{ attribute 'TcHmiSymbol.AddSymbol' }
	MS7 : ST_DeviceDualChannelInput;
	
	
	//ACCESS POINT Devices
	{ attribute 'TcHmiSymbol.AddSymbol' }
	LC1 : ST_DeviceDualChannelInput;
	{ attribute 'TcHmiSymbol.AddSymbol' }
	LC2 : ST_DeviceDualChannelInput;
	{ attribute 'TcHmiSymbol.AddSymbol' }
	LC3 : ST_DeviceDualChannelInput;
	{ attribute 'TcHmiSymbol.AddSymbol' }
	GS1 : ST_DeviceDualChannelInput;
	
	//Misc devices
	{ attribute 'TcHmiSymbol.AddSymbol' }
	PendantEnable : ST_DeviceDualChannelInput;
	{ attribute 'TcHmiSymbol.AddSymbol' }
	SearchAndLock : ST_DeviceDualChannelInput;
	{ attribute 'TcHmiSymbol.AddSymbol' }
	Hmi_Maintenance  : ST_DeviceDualChannelInput;
	
	Q1Q2 AT %I* : BOOL;
	Q3Q4 AT %I* : BOOL;
	SPB1 AT %I* : BOOL;
	SPB2 AT %I* : BOOL;
	HmiRb AT %I* : BOOL;
	HmiLocal AT %I* : BOOL;
	HmiNormal AT %I* : BOOL;
	
	//Status Signals
	EstopsHealthy AT %I* : BOOL;
	inMode_Maintenance AT %I* : BOOL;
	inMode_Local AT %I* : BOOL;
	inMode_Normal AT %I* : BOOL;
	inMode_SearchedAndLocked AT %I* : BOOL;
	
	IncidentSlitsSwitch AT %I* : BOOL;
	
	
	SampleAreaSearched_Downstream AT %I* : BOOL;
	SampleAreaSearched_Upstream AT %I* : BOOL;
	
	SampleStackZRotationSLSHealthy AT %I* : BOOL;
	
	EDMErr_NonSampleArea AT %I* : BOOL;
	EDMErr_SampleArea AT %I* : BOOL;
	
	upstreamSearchReq : BOOL;
	downstreamSearchReq : BOOL;
	
	//Pendant statuses
	AccessPointCrossed AT %I* : BOOL;
	AccessPointsMuted AT %I* : BOOL;
	PendantMuted AT %I* : BOOL;
	SLS_Muted AT %I* : BOOL;
	
	//Maintenance muting
	Mute_AccessPoints AT %Q* : BOOL;
	Mute_PendantEnable AT %Q* : BOOL;
	Mute_SLS AT %Q* : BOOL;
	
	
	
	
	
	SAMPLE_MOTION_PERMIT AT %I* : BOOL; //signal from the sto control to send a stop command
	MOTION_PERMIT AT %I* : BOOL;	//Not in use?
	NON_SAMPLE_MOTION_PERMIT  AT %I* : BOOL;
	
	MotionIsolator AT %I* : BOOL; //Physical isolator on side of panel
	
	
	
	
	
	
	//Output Devices
	Q1 AT %I* : BOOL;
	Q2 AT %I* : BOOL;
	Q3 AT %I* : BOOL;
	Q4 AT %I* : BOOL;
	SB1 AT %I* : BOOL;
	SB2 AT %I* : BOOL;
	MSS1_1 AT %I* : BOOL;
	MSS1_2 AT %I* : BOOL;
	MSS2_1 AT %I* : BOOL;
	MSS2_2 AT %I* : BOOL;
	MSS3_1 AT %I* : BOOL;
	MSS3_2 AT %I* : BOOL;
	RCU AT %I* : BOOL;
	HmiRbLight AT %I* : BOOL;
	HmiTripped AT %I* : BOOL;
	HmiMaintenance AT %I* : BOOL;
	
	//Physical input device
	HMI_ErrorAckButton AT %I* : BOOL;
	ErrorAckLightState : BOOL;
	HMI_ErrorAckLight AT %Q* : BOOL;
	HMI_SafetyRunLight AT %Q* : BOOL;
	
	lostSamplePermit : F_TRIG;
	lostNonSamplePermit : F_TRIG;
	gotSamplePermit : R_TRIG;
	gotNonSamplePermit : R_TRIG;
	//screen blackout
	fbStartWindowsCommand : NT_StartProcess; // Start Windows Command
	sPath : T_MaxString := 'C:\Windows\System32\cmd.exe' ;
	sDirName : T_MaxString := 'C:\Windows\System32' ;
	sCommandLine : T_MaxString := 'cmd /c scrnsave.scr /s'; 
	bStartWindowsCommand : BOOL;
	searchRTrig : R_TRIG;
	collisionDetectedRTrig : R_Trig;
	maintenanceAllowRemote : BOOL:= FALSE;
	
END_VAR
VAR_OUTPUT
	STOP_MOTION : BOOL;
	NON_SAMPLE_PERMIT : BOOL;
	SAMPLE_PERMIT : BOOL;
	STOP_NON_SAMPLE_MOTION : BOOL;
	SAMPLE_PERMIT_R_EDGE : BOOL;
	NON_SAMPLE_PERMIT_R_EDGE : BOOL;
	inLocalMode : BOOL;
	CollisionDetected : BOOL;
	collisionDetected_R_Edge : BOOL;
END_VAR

inLocalMode := inMode_Local OR inMode_Maintenance;
ERRACK := HMI_ErrorAckButton;

lostSamplePermit(CLK:= SAMPLE_MOTION_PERMIT);
STOP_MOTION:= lostSamplePermit.Q;
lostNonSamplePermit(CLK:= NON_SAMPLE_MOTION_PERMIT);
STOP_NON_SAMPLE_MOTION:= lostNonSamplePermit.Q;
NON_SAMPLE_PERMIT := NON_SAMPLE_MOTION_PERMIT;
SAMPLE_PERMIT := SAMPLE_MOTION_PERMIT;

gotSamplePermit(CLK:= SAMPLE_MOTION_PERMIT);
gotNonSamplePermit(CLK:=NON_SAMPLE_MOTION_PERMIT);
SAMPLE_PERMIT_R_EDGE:= gotSamplePermit.Q;
NON_SAMPLE_PERMIT_R_EDGE:= gotNonSamplePermit.Q;

CollisionDetected := NOT IncidentSlitsSwitch;
collisionDetectedRTrig(Clk:=CollisionDetected);
collisionDetected_R_Edge:= collisionDetectedRTrig.Q;

IF NOT inMode_Maintenance THEN
	Mute_AccessPoints := FALSE;
	Mute_PendantEnable := FALSE;
END_IF
FOR i:=1 TO 7 DO
	SafetyTargets[i].Diag:=0;
	SafetyTargets[i].State:=1;
	FOR j:=1 TO 10 DO
		IF SafetyTargets[i].aSafetyGroups[j].Connected THEN
			IF SafetyTargets[i].aSafetyGroups[j].STATE <> 1 THEN
				SafetyTargets[i].State:=SafetyTargets[i].aSafetyGroups[j].STATE;
				SafetyTargets[i].Diag:=SafetyTargets[i].aSafetyGroups[j].DIAG;
				EXIT;
			END_IF
		END_IF			
	END_FOR
	
	CASE SafetyTargets[i].Diag OF
		0:	SafetyTargets[i].Diag_String:= 'No Error';
		1:	SafetyTargets[i].Diag_String:= 'FB Error';
		2:	SafetyTargets[i].Diag_String:= 'Comm Error';
		3:	SafetyTargets[i].Diag_String:= 'Module Error';
		4:	SafetyTargets[i].Diag_String:= 'CMP Error';
		5:	SafetyTargets[i].Diag_String:= 'Deactive';
		6:	SafetyTargets[i].Diag_String:= 'Restart Error';
	END_CASE
	CASE SafetyTargets[i].State OF
		1: SafetyTargets[i].State_String:= 'Run';
		2: SafetyTargets[i].State_String:= 'Stop';
		4: SafetyTargets[i].State_String:= 'Error';
		5: SafetyTargets[i].State_String:= 'Reset';
		6: SafetyTargets[i].State_String:= 'Start';
		7: SafetyTargets[i].State_String:= 'Stop Err';
		16: SafetyTargets[i].State_String:= 'Deactive';
		17: SafetyTargets[i].State_String:= 'Wait Comm Err';
	END_CASE
END_FOR

//Error ack light
ErrorAckLightState:= FALSE;
IF NOT inMode_SearchedAndLocked THEN	//We don't turn on light in S&L
	FOR i:=1 TO 7 DO
		IF SafetyTargets[i].State <> 1 THEN
			ErrorAckLightState:= TRUE;
		END_IF
	END_FOR
END_IF

HMI_ErrorAckLight := ErrorAckLightState;
HMI_SafetyRunLight := RUN AND NOT inMode_SearchedAndLocked;

//Blackout screen
searchRTrig(CLK:= inMode_SearchedAndLocked);
bStartWindowsCommand:= searchRTrig.Q;
fbStartWindowsCommand(
        NETID:= '', 
        PATHSTR:= sPath, 
        DIRNAME:= sDirName, 
        COMNDLINE:= sCommandLine, 
        START:= bStartWindowsCommand, 
        TMOUT:= T#5S, 
        BUSY=> , 
        ERR=> , 
        ERRID=> );

IF inMode_Normal THEN
	IF NOT SampleAreaSearched_Downstream THEN
		downstreamSearchReq := TRUE;
	ELSE
		downstreamSearchReq := FALSE;
	END_IF
	IF NOT SampleAreaSearched_Upstream THEN
		upstreamSearchReq := TRUE;
	ELSE
		upstreamSearchReq := FALSE;
	END_IF
ELSE
	upstreamSearchReq := FALSE;
	downstreamSearchReq := FALSE;
END_IF

//Banner message logic
IF SafetyTargets[1].State = 4 THEN
	BannerMessage:= 'Safety in error';
ELSIF SafetyTargets[1].State <> 1 THEN
	BannerMessage:= 'EL6910 Safety not running';
ELSIF SafetyTargets[2].State <>1 OR SafetyTargets[3].State <> 1 OR SafetyTargets[4].State <> 1 OR SafetyTargets[5].State <> 1 OR SafetyTargets[6].State <> 1 OR SafetyTargets[7].State <> 1 THEN
	BannerMessage:= 'Drive safety project not running';
ELSIF NOT EstopsHealthy  THEN
	BannerMessage:= 'Estop pressed';
ELSIF NOT LC1.Output THEN
	BannerMessage:= 'LC1 access point not healthy';
ELSIF NOT LC2.Output THEN
	BannerMessage:= 'LC2 access point not healthy';
ELSIF NOT LC3.Output THEN
	BannerMessage:= 'LC3 access point not healthy';
ELSIF NOT GS1.Output THEN
	BannerMessage:= 'GS1 access point not healthy';	
ELSIF NOT SampleStackZRotationSLSHealthy THEN
	BannerMessage:= 'Sample stack rotation SLS tripped';
ELSIF HmiRbLight THEN
	BannerMessage:= 'Reset required';
ELSIF upstreamSearchReq AND downstreamSearchReq AND inMode_Normal THEN
	BannerMessage:= 'Sample area upstream and downstream require search';
ELSIF upstreamSearchReq AND inMode_Normal THEN
	BannerMessage:= 'Sample area upstream requires search';
ELSIF downstreamSearchReq AND inMode_Normal THEN
	BannerMessage:= 'Sample area downstream requires search';
ELSIF inMode_Local THEN
	BannerMessage:= 'Only control from pendant permitted';
ELSIF inMode_Normal AND CollisionDetected THEN
	BannerMessage:= 'Collision detected, control only possible in local mode';
ELSE
	BannerMessage:= '';
END_IF

END_PROGRAM

// ---- POUs/Application_Specific/Applications/Pendant.TcPOU
PROGRAM Pendant
VAR
	astHmiControl: ARRAY [1..GVL_APP.nAXIS_NUM] OF ST_PendantControl;
	eHmiControl : E_PendantControl;
	eSWLimitControl : E_SWLimitControl;
	iHmiAxisSelection : INT;
	iKeyPressedValue : INT := -1;
	iSelectedAxis : INT := -1;
	aiUsedKeys : ARRAY[1..12] OF INT := [E_PendantControl.JogFwd, E_PendantControl.JogBwd,
    E_PendantControl.SmallTweakFwd, E_PendantControl.SmallTweakBwd, E_PendantControl.MediumTweakFwd, 
	E_PendantControl.MediumTweakBwd, E_PendantControl.BigTweakFwd, E_PendantControl.BigTweakBwd, 
	E_PendantControl.AbsMove, E_PendantControl.Stop, E_PendantControl.SlowJogFwd, E_PendantControl.SlowJogBwd];
	iUsedKeysIndex : INT;
	iSmallTweakDistance : REAL := 0.1;	
	iMediumTweakDistance : REAL := 1;
	iBigTweakDistance : REAL := 5;
	iHmiAxisCounter : INT;
	bResetParameters : BOOL := FALSE;
	
	bLocalMode: BOOL;
	fbLocalModeRTrig: R_TRIG;
	fbLocalModeFTrig: F_TRIG;
	
	bSWLimitsOn : BOOL := FALSE; //False for off, true for on
END_VAR

bLocalMode:= SAFETY.inLocalMode;
fbLocalModeRTrig(CLK := bLocalMode);
fbLocalModeFTrig(CLK := bLocalMode);

IF bResetParameters THEN
	ResetParameters();
END_IF


IF ketop.keys[E_PendantControl.Stop] OR NOT bLocalMode THEN
	eHmiControl := E_PendantControl.Stop;
END_IF


CASE eHmiControl OF
	E_PendantControl.Default:
		iKeyPressedValue := -1;
		iSelectedAxis := -1;
		IF iHmiAxisSelection > 0 AND iHmiAxisSelection <= UINT_TO_INT(GVL_APP.nAXIS_NUM) THEN
			FOR iUsedKeysIndex := 1 TO (SIZEOF(aiUsedKeys)/SIZEOF(UINT)) DO
				IF KeTop.keys[aiUsedKeys[iUsedKeysIndex]] = TRUE THEN
					iKeyPressedValue := aiUsedKeys[iUsedKeysIndex];
					iSelectedAxis := iHmiAxisSelection;
					eHmiControl := iKeyPressedValue;
				END_IF
			END_FOR
		END_IF
		
	E_PendantControl.JogFwd:
		astAxes[iSelectedAxis].stControl.fVelocity := ABS(astAxes[iSelectedAxis].stControl.fVelocity);
		Jog();
		eHmiControl := E_PendantControl.WaitForJogFinish;
	
	E_PendantControl.JogBwd:
		astAxes[iSelectedAxis].stControl.fVelocity := -ABS(astAxes[iSelectedAxis].stControl.fVelocity);
		Jog();
		eHmiControl := E_PendantControl.WaitForJogFinish;	
		
	E_PendantControl.SlowJogFwd:
		astAxes[iSelectedAxis].stControl.fVelocity := ABS(astAxes[iSelectedAxis].stControl.fVelocity);
		SlowJog();
		eHmiControl := E_PendantControl.WaitForJogFinish;		
		
	E_PendantControl.SlowJogBwd:
		astAxes[iSelectedAxis].stControl.fVelocity := -ABS(astAxes[iSelectedAxis].stControl.fVelocity);
		SlowJog();
		eHmiControl := E_PendantControl.WaitForJogFinish;		
		
	E_PendantControl.WaitForJogFinish:
		IF Ketop.keys[iKeyPressedValue] = FALSE THEN
			astAxes[iSelectedAxis].stControl.bHalt := TRUE;
			eHmiControl := E_PendantControl.Default;
		END_IF

	E_PendantControl.SmallTweakFwd:
		astAxes[iSelectedAxis].stControl.fRelativePosition := ABS(iSmallTweakDistance);
		Tweak();
		eHmiControl := E_PendantControl.WaitForTweakFinish;

	E_PendantControl.SmallTweakBwd:
		astAxes[iSelectedAxis].stControl.fRelativePosition := -ABS(iSmallTweakDistance);
		Tweak();
		eHmiControl := E_PendantControl.WaitForTweakFinish;
	
	E_PendantControl.MediumTweakFwd:
		astAxes[iSelectedAxis].stControl.fRelativePosition := ABS(iMediumTweakDistance);
		Tweak();
		eHmiControl := E_PendantControl.WaitForTweakFinish;

	E_PendantControl.MediumTweakBwd:
		astAxes[iSelectedAxis].stControl.fRelativePosition := -ABS(iMediumTweakDistance);
		Tweak();
		eHmiControl := E_PendantControl.WaitForTweakFinish;
		
	E_PendantControl.BigTweakFwd:
		astAxes[iSelectedAxis].stControl.fRelativePosition := ABS(iBigTweakDistance);
		Tweak();
		eHmiControl := E_PendantControl.WaitForTweakFinish;

	E_PendantControl.BigTweakBwd:
		astAxes[iSelectedAxis].stControl.fRelativePosition := -ABS(iBigTweakDistance);
		Tweak();
		eHmiControl := E_PendantControl.WaitForTweakFinish;
		
	E_PendantControl.WaitForTweakFinish:
		IF Ketop.keys[iKeyPressedValue] = FALSE AND astAxes[iSelectedAxis].stStatus.bMoving = FALSE THEN
			eHmiControl := E_PendantControl.Default;
		END_IF
		
	E_PendantControl.AbsMove:
		astAxes[iSelectedAxis].stConfig.fOverride := astHmiControl[iSelectedAxis].fVelocity;
		astAxes[iSelectedAxis].stControl.fPosition := astHmiControl[iSelectedAxis].fTargetPosition;
		astAxes[iSelectedAxis].stControl.eCommand := E_MotionFunctions.eLocalMoveAbsolute;
		astAxes[iSelectedAxis].stControl.bExecute := TRUE; 
		eHmiControl := E_PendantControl.WaitForAbsoluteFinish;
	
	E_PendantControl.WaitForAbsoluteFinish:
		IF astAxes[iSelectedAxis].stStatus.bMoving = FALSE THEN
			eHmiControl := E_PendantControl.Default;	
		END_IF
	
	E_PendantControl.Stop:
		IF iSelectedAxis > 0 THEN
			astAxes[iSelectedAxis].stControl.bHalt := TRUE;
			IF ketop.keys[E_PendantControl.Stop] = FALSE AND astAxes[iSelectedAxis].stStatus.bMoving = FALSE THEN
				eHmiControl := E_PendantControl.Default;
				FOR iUsedKeysIndex := 1 TO (SIZEOF(aiUsedKeys)/SIZEOF(UINT)) DO
					IF KeTop.keys[aiUsedKeys[iUsedKeysIndex]] = TRUE THEN
						eHmiControl := E_PendantControl.Stop;
					END_IF
				END_FOR
			END_IF	
		END_IF
		IF iSelectedAxis = -1 AND bLocalMode THEN
			eHmiControl := E_PendantControl.Default;
		END_IF

END_CASE

CASE eSWLimitControl OF
	E_SWLimitControl.Default:
		IF fbLocalModeRTrig.Q THEN
			//eSWLimitControl := E_SWLimitControl.EnableSWLimits;
		END_IF
		IF fbLocalModeFTrig.Q THEN
			eSWLimitControl := E_SWLimitControl.DisableSWLimits;
		END_IF
	
	E_SWLimitControl.EnableSWLimits:
		bSWLimitsOn := TRUE;
		KeTop.screenBrightness := 100;
		FOR iHmiAxisCounter := 1 TO GVL_APP.nAXIS_NUM DO
			ToggleSWLimits();	
		END_FOR
		eSWLimitControl := E_SWLimitControl.Default;
	
	E_SWLimitControl.DisableSWLimits:
		bSWLimitsOn := FALSE;
		FOR iHmiAxisCounter := 1 TO GVL_APP.nAXIS_NUM DO
			ToggleSWLimits();	
		END_FOR
		eSWLimitControl := E_SWLimitControl.Default;
	
	E_SWLimitControl.WriteFwdLimit:
		IF bLocalMode THEN
			astAxes[iHmiAxisSelection].stConfig.eAxisParameters := E_AxisParameters.SWLimitForward;
			astAxes[iHmiAxisSelection].stConfig.fWriteAxisParameter := astHmiControl[iHmiAxisSelection].fFwdLimit;
			WriteToSWLimit();
		END_IF
		eSWLimitControl := E_SWLimitControl.Default;
	
	E_SWLimitControl.WriteBwdLimit:
		IF bLocalMode THEN
			astAxes[iHmiAxisSelection].stConfig.eAxisParameters := E_AxisParameters.SWLimitBackward;
			astAxes[iHmiAxisSelection].stConfig.fWriteAxisParameter := astHmiControl[iHmiAxisSelection].fBwdLimit;
			WriteToSWLimit();	
		END_IF
		eSWLimitControl := E_SWLimitControl.Default;
	
END_CASE

ACTION Jog:
astAxes[iSelectedAxis].stConfig.fOverride := 100;
astAxes[iSelectedAxis].stControl.eCommand:= E_MotionFunctions.eLocalMoveVelocity;
astAxes[iSelectedAxis].stControl.bExecute:= TRUE;
END_ACTION

ACTION ResetParameters:
FOR iHmiAxisCounter := 1 TO GVL_APP.nAXIS_NUM DO
	astHmiControl[iHmiAxisCounter].fTargetPosition := 0;
	astHmiControl[iHmiAxisCounter].fVelocity := 100;	
END_FOR
bResetParameters := FALSE;
END_ACTION

ACTION SlowJog:
astAxes[iSelectedAxis].stConfig.fOverride := 20;
astAxes[iSelectedAxis].stControl.eCommand:=E_MotionFunctions.eLocalMoveVelocity;
astAxes[iSelectedAxis].stControl.bExecute:= TRUE;
END_ACTION

ACTION ToggleSWLimits:
astAxes[iHmiAxisCounter].stControl.eCommand := E_MotionFunctions.eWriteToggleSWLimits;
astAxes[iHmiAxisCounter].stConfig.fWriteAxisBoolParameter := bSWLimitsOn;
astAxes[iHmiAxisCounter].stControl.bExecute := TRUE;
END_ACTION

ACTION Tweak:
astAxes[iSelectedAxis].stConfig.fOverride :=100;
astAxes[iSelectedAxis].stControl.eCommand:=E_MotionFunctions.eLocalMoveRelative;
astAxes[iSelectedAxis].stControl.bExecute:=TRUE;
END_ACTION

ACTION WriteToSWLimit:
astAxes[iHmiAxisSelection].stControl.eCommand := E_MotionFunctions.eWriteParameter;
astAxes[iHmiAxisSelection].stControl.bExecute := TRUE;
END_ACTION

END_PROGRAM

// ---- POUs/PANEL.TcPOU
PROGRAM PANEL
VAR
	//ECB1 : ST_ECB:= (Name:= 'MSR', Description:= 'Safety devices');
	//ECB2 : ST_ECB:= (Name:= 'MR1-control', Description:= '24V Axes 1-8'); //MR1
END_VAR

END_PROGRAM

// ---- POUs/Application_Specific/Axes/Axis_Template.TcPOU
PROGRAM Axis_Template
VAR
	iAxisNumber : INT := E_AxisNames.Axis1;
	iGroupNumber : INT := 1;
	
	stoRTrig : R_Trig;
	
	//Automatic reset on permit
	startReset : BOOL;
	resetDelay : TON;
	startDisable : BOOL;
	disableDelay : TON;
END_VAR

//Initial parameters of an Axis
(*
IF _TaskInfo[fbGetCurTaskIndex.index].FirstCycle THEN
    //Initial default values:
    GVL.astAxes[iAxisNumber].stHomingConfig.eHomeSeq :=E_HomingRoutines.eHomeToEncPulse_viaBwdLimit;
	GVL.astAxes[iAxisNumber].stHomingConfig.fHomeAbsPosition:= 0;
	GVL.astAxes[iAxisNumber].stHomingConfig.fHomeMidRelativeMove:=1;
    GVL.astAxes[iAxisNumber].stHomingConfig.fHomePosition := 0;
    GVL.astAxes[iAxisNumber].stHomingConfig.fHomeFinishDistance := 0.0;
    GVL.astAxes[iAxisNumber].stConfig.eRestorePosition := E_RestorePosition.eRestoreWithoutHome;
	GVL.astAxes[iAxisNumber].stControl.bAutoEnableDisable := TRUE;
	GVL.astAxes[iAxisNumber].stControl.tMoveFinishedDelay := T#0.1S;
	//Set which group this axis belongs to
	GVL.astAxes[iAxisNumber].stDescription.iGroupNumber := iGroupNumber;
	GVL.astAxes[iAxisNumber].Commissioning := FALSE;
	GVL.astAxes[iAxisNumber].stDescription.sUnits:= 'mm';
END_IF

//Permit
GVL.astAxes[iAxisNumber].stInputs.bPermit := TRUE;//(SAFETY.SAMPLE_PERMIT AND NOT SAFETY.CollisionDetected) OR (SAFETY.SAMPLE_PERMIT AND (safety.inMode_Local OR safety.inMode_Maintenance));

//Remote operation toggle

IF SAFETY.inMode_Local THEN
	GVL.astAxes[iAxisNumber].stInputs.bAllowRemoteControl:= FALSE;
ELSIF SAFETY.inMode_Maintenance AND NOT SAFETY.maintenanceAllowRemote THEN
	GVL.astAxes[iAxisNumber].stInputs.bAllowRemoteControl:= FALSE;
ELSE
	GVL.astAxes[iAxisNumber].stInputs.bAllowRemoteControl:= TRUE;
END_IF

//Do an automatic reset on regaining permit;

IF SAFETY.SAMPLE_PERMIT_R_EDGE THEN
	startReset:= TRUE;
END_IF
resetDelay(IN:= startReset, PT:= T#0.5S);
IF resetDelay.Q THEN
	startReset := FALSE;
	GVL.astAxes[iAxisNumber].stControl.bReset:= TRUE;
END_IF


//Disable axis if no permit

IF SAFETY.STOP_MOTION THEN
	startDisable := TRUE;
END_IF
disableDelay(IN:= startDisable, PT:= T#1S);
IF disableDelay.Q THEN
	startDisable:= FALSE;
	GVL.astAxes[iAxisNumber].stControl.bEnable:= FALSE;
END_IF



//Safety stop motion

IF SAFETY.STOP_MOTION THEN
	GVL.astAxes[iAxisNumber].stControl.bHalt:= TRUE;
END_IF
IF SAFETY.collisionDetected_R_Edge THEN
	GVL.astAxes[iAxisNumber].stControl.bHalt:= TRUE;
END_IF

stoRTrig(CLK:=GVL.astAxes[iAxisNumber].stStatus.bSTOActive);
IF stoRTrig.Q THEN
	GVL.astAxes[iAxisNumber].stControl.bReset:= TRUE;
END_IF
*)

END_PROGRAM

// ---- POUs/Application_Specific/Groups/GROUP_1.TcPOU
PROGRAM GROUP_1
VAR
	iSetGroupNumber : INT := 1; //SET THIS TO THE NUMBER FOR THIS GROUP
END_VAR

IF _TaskInfo[fbGetCurTaskIndex.index].FirstCycle THEN
	GVL.iAxesGroupIndex := 1;
	FOR GVL.iAxis := 1 TO GVL_APP.nAXIS_NUM DO
		IF astAxes[GVL.iAxis].stDescription.iGroupNumber = iSetGroupNumber THEN
			GVL.astAxesGroup[iSetGroupNumber].aAxesInGroup[GVL.iAxesGroupIndex] := UINT_TO_INT(GVL.iAxis);
			GVL.iAxesGroupIndex := GVL.iAxesGroupIndex + 1;
		END_IF
	END_FOR
	GVL.astAxesGroup[iSetGroupNumber].stDescription.iAxesInGroup := GVL.iAxesGroupIndex -1;
END_IF

END_PROGRAM

// ---- POUs/Application_Specific/Groups/Group_Template.TcPOU
PROGRAM Group_Template
VAR
	//iSetGroupNumber : INT := 1; //SET THIS TO THE NUMBER FOR THIS GROUP
END_VAR

//Sample code for defining groups by iterating through each axis on startup and adding all matching axis to this array
(*
IF _TaskInfo[fbGetCurTaskIndex.index].FirstCycle THEN
	GVL.iAxesGroupIndex := 1;
	FOR GVL.iAxis := 1 TO GVL_APP.nAXIS_NUM DO
		IF astAxes[GVL.iAxis].stDescription.iGroupNumber = iSetGroupNumber THEN
			GVL.astAxesGroup[iSetGroupNumber].aAxesInGroup[GVL.iAxesGroupIndex] := UINT_TO_INT(GVL.iAxis);
			GVL.iAxesGroupIndex := GVL.iAxesGroupIndex + 1;
		END_IF
	END_FOR
	GVL.astAxesGroup[iSetGroupNumber].stDescription.iAxesInGroup := GVL.iAxesGroupIndex -1;
END_IF
*)

END_PROGRAM

// ---- tc_mca_std_lib/POUs/Motion/FB_AxisGroups.TcPOU
FUNCTION_BLOCK FB_AxisGroups
VAR_INPUT
END_VAR
VAR_OUTPUT
END_VAR
VAR
	_stAxisGroup: REFERENCE TO ST_AxisGroupStruct;
	iGroupedAxis : INT;
END_VAR

METHOD mStatus_GroupEnabled : BOOL
VAR_INPUT
END_VAR
_stAxisGroup.stFlag.iDisabled := 0;
_stAxisGroup.stFlag.bDisabledFlag := FALSE;
_stAxisGroup.stFlag.iNumberOfAxisDisabled := 0;
FOR iGroupedAxis := 1 TO GVL.nMAX_AXES_PER_GROUP DO
	IF _stAxisGroup.aAxesInGroup[iGroupedAxis] = 0 THEN
		IF _stAxisGroup.stFlag.iDisabled <> 0 THEN
			_stAxisGroup.stFlag.bDisabledFlag := TRUE;	
		END_IF
		RETURN;
	END_IF
	_stAxisGroup.stFlag.iDisabled := _stAxisGroup.stFlag.iDisabled + BOOL_TO_INT(NOT astAxes[_stAxisGroup.aAxesInGroup[iGroupedAxis]].stStatus.bEnabled) * iGroupedAxis;
	_stAxisGroup.stFlag.iNumberOfAxisDisabled := _stAxisGroup.stFlag.iNumberOfAxisDisabled + BOOL_TO_INT(NOT astAxes[_stAxisGroup.aAxesInGroup[iGroupedAxis]].stStatus.bEnabled);
END_FOR
END_METHOD

METHOD mStatus_GroupError : BOOL
VAR_INPUT
END_VAR
_stAxisGroup.stFlag.iError := 0;
_stAxisGroup.stFlag.bErrorFlag := FALSE;
_stAxisGroup.stFlag.iNumberOfAxisInError := 0; 

FOR iGroupedAxis := 1 TO GVL.nMAX_AXES_PER_GROUP DO
	IF _stAxisGroup.aAxesInGroup[iGroupedAxis] = 0 THEN
		IF _stAxisGroup.stFlag.iError <> 0 THEN
			_stAxisGroup.stFlag.bErrorFlag := TRUE;
		END_IF
		RETURN;
	END_IF
	_stAxisGroup.stFlag.iError := _stAxisGroup.stFlag.iError + BOOL_TO_INT(astAxes[_stAxisGroup.aAxesInGroup[iGroupedAxis]].stStatus.bError) * (100 + iGroupedAxis);
	_stAxisGroup.stFlag.iNumberOfAxisInError := _stAxisGroup.stFlag.iNumberOfAxisInError + BOOL_TO_INT(astAxes[_stAxisGroup.aAxesInGroup[iGroupedAxis]].stStatus.bError);
END_FOR
END_METHOD

METHOD mStatus_GroupState : BOOL
VAR_INPUT
END_VAR
_stAxisGroup.stFlag.iState := _stAxisGroup.stFlag.iDisabled + _stAxisGroup.stFlag.iError;
END_METHOD

METHOD Run : BOOL
VAR_INPUT
END_VAR
mStatus_GroupEnabled();
mStatus_GroupError();
mStatus_GroupState();
END_METHOD

PROPERTY stAxisGroup : REFERENCE TO ST_AxisGroupStruct
GET
stAxisGroup REF= _stAxisGroup;
END_GET
SET
_stAxisGroup REF= stAxisGroup;
END_SET
END_PROPERTY

END_FUNCTION_BLOCK

// ---- tc_mca_std_lib/POUs/Motion/FB_SlitPair.TcPOU

FUNCTION_BLOCK FB_SlitPair
VAR_INPUT
    iBladeNegative: UINT; //Axis ID for negatively positioned blade
    iBladePositive: UINT; //Axis ID for positively positioned blade
    iGapSize: UINT; //Axis ID for the size of gap between slit blades
    iGapCentre: UINT; //Axis ID for the centre position of the gap formed by slit blades
    bEnable: BOOL; //Enable/disable the slit set
    bReset: BOOL; //Reset the slit set
    fEncoderScaling: LREAL := 10000; //default scaling denominator of 10000
    bAutoHome: BOOL := FALSE;
END_VAR
VAR_OUTPUT
    bEnabled: BOOL := FALSE; //Enabled status of function
    bError: BOOL; //Error status of function
    bHoming: BOOL := FALSE; //TRUE if function is homing axes
END_VAR
VAR
    eSlitPairState: E_SlitPairStates := E_SlitPairStates.INIT; //statemachine index

//Internal statuses for logic
    bResetting: BOOL := FALSE; //TRUE if axis going through a reset
    bAxesEnabled: BOOL := FALSE; //TRUE if all axes enabled
    bBladesHomed: BOOL:= FALSE; //TRUE if blade axes are calibrated
    bGapHomed: BOOL:= FALSE; //TRUE if virtual axes are calibrated
    bBladesCoupled: BOOL:= FALSE; //TRUE if both blade axes are coupled
    bBladesUncoupled: BOOL := FALSE; //TRUE if both blade axes are uncoupled
    bAxisErrorsPresent: BOOL := FALSE; //TRUE if error present on any real or virtual axis
    bFunctionInErrorState: BOOL := FALSE; //TRUE if function block is in one of the error related states
    fGapSizePosition: LREAL;
    iGapSizePosition AT %Q*: UDINT := 0;
    fGapCentrePosition: LREAL;
    iGapCentrePosition AT %Q*: UDINT := 0;
    resetCounterTimeout: UINT :=0;
    mcHomeGapSize: MC_Home;
    mcHomeGapCentre: MC_Home;
END_VAR


(* NOTES
For the virtual axis setup, the encoders need their type changed from "simulation encoder" to "Encoder (Universal)".
In addition the scale factor needs to be changed to a numerator of 1 and denominator of fEncoderScaling which is 10,000 by default)
Care needs to be taken with scaling and setup of both real and virtual axes to ensure velocities are not too fast and axes have time to settle before they submit a "complete move"
*)

//Configure homing routine of virtual axes
GVL.astAxes[iGapSize].stConfig.eHomeSeq := E_HomingRoutines.eHomeDirect;
GVL.astAxes[iGapCentre].stConfig.eHomeSeq := E_HomingRoutines.eHomeDirect;

//Run actions for slit set
actErrorHandling(); //Error handling subroutine
actGapLimits(); //Set virtual axis limits to TRUE
actVirtualAxisPositions(); //Virtual axis encoder position subroutine
actRunMethods(); //Update statuses

//Mc_Home FBs configured to clear homing signal
mcHomeGapSize(Axis := astAxes[iGapSize].Axis, HomingMode:=MC_HomingMode.MC_ResetCalibration);
mcHomeGapCentre(Axis:=astAxes[iGapCentre].Axis, HomingMode:=MC_HomingMode.MC_ResetCalibration);
mcHomeGapSize.Execute := FALSE;
mcHomeGapCentre.Execute := FALSE;

CASE eSlitPairState OF
    E_SlitPairStates.INIT:
        IF bAxesEnabled AND bEnable THEN
            eSlitPairState := E_SlitPairStates.INIT_CLEAR_GEARING;
        END_IF

    E_SlitPairStates.INIT_CLEAR_GEARING:
        actClearSlitGearing();
        eSlitPairState := E_SlitPairStates.INIT_GEAROUT_CHECK;

    E_SlitPairStates.INIT_GEAROUT_CHECK: //Check gearOut completion
        IF bBladesUncoupled THEN
            eSlitPairState := E_SlitPairStates.CHECK_HOME_STATUS;
        END_IF

    E_SlitPairStates.CHECK_HOME_STATUS: //If blades are already homed, skip to virtual homing, if blades not homed and autohome enabled then home blades, otherwise wait for blades to be homed
        IF bBladesHomed THEN
            eSlitPairState := E_SlitPairStates.HOME_GAP; //Skip to functioning
        ELSIF bAutoHome THEN
            eSlitPairState := E_SlitPairStates.HOME_BLADES; //If autohome enabled, home the blades
        END_IF

    E_SlitPairStates.HOME_BLADES: //Initiate homing of blade axes. Homing routine must be pre-configured by user
        GVL.astAxes[iBladeNegative].stControl.eCommand := E_MotionFunctions.eHome;
        GVL.astAxes[iBladePositive].stControl.eCommand := E_MotionFunctions.eHome;
        GVL.astAxes[iBladeNegative].stControl.bExecute := TRUE;
        GVL.astAxes[iBladePositive].stControl.bExecute := TRUE;
        bHoming := TRUE;
        eSlitPairState := E_SlitPairStates.CHECK_BLADE_HOME_COMPLETE;

    E_SlitPairStates.CHECK_BLADE_HOME_COMPLETE: //Wait for completion of blade homing routines
        IF bBladesHomed THEN
            eSlitPairState := E_SlitPairStates.HOME_GAP;
            bHoming := FALSE;
        END_IF

    E_SlitPairStates.HOME_GAP: //"Home" the virtual axes
        GVL.astAxes[iGapSize].stConfig.eHomeSeq := E_HomingRoutines.eHomeDirect;
        GVL.astAxes[iGapCentre].stConfig.eHomeSeq := E_HomingRoutines.eHomeDirect;
        GVL.astAxes[iGapSize].stConfig.fHomePosition := fGapSizePosition;
        GVL.astAxes[iGapCentre].stConfig.fHomePosition := fGapCentrePosition;
        GVL.astAxes[iGapSize].stControl.eCommand := E_MotionFunctions.eHome;
        GVL.astAxes[iGapCentre].stControl.eCommand := E_MotionFunctions.eHome;
        GVL.astAxes[iGapSize].stControl.bExecute := TRUE;
        GVL.astAxes[iGapCentre].stControl.bExecute := TRUE;
        eSlitPairState := E_SlitPairStates.CHECK_GAP_HOME_COMPLETE;

    E_SlitPairStates.CHECK_GAP_HOME_COMPLETE: //Wait for virtual homing completion
        IF bGapHomed THEN
            eSlitPairState := E_SlitPairStates.GEARIN_SLITS;
        END_IF

    E_SlitPairStates.GEARIN_SLITS: //Setup gearing
        actSetupSlitGearing();
        eSlitPairState := E_SlitPairStates.CHECK_GEARIN_SLITS_COMPLETE;

    E_SlitPairStates.CHECK_GEARIN_SLITS_COMPLETE: //Wait for gearing complete
        IF bBladesCoupled THEN
            eSlitPairState := E_SlitPairStates.SLITS_OPERATIONAL;
        END_IF

    E_SlitPairStates.SLITS_OPERATIONAL: //SLITS OPERATIONAL - Monitor for any gear outs and re-gear when no busy blades
        bEnabled := TRUE;
        IF NOT bBladesCoupled AND NOT GVL.astAxes[iBladeNegative].stStatus.bBusy AND NOT GVL.astAxes[iBladePositive].stStatus.bBusy THEN
            eSlitPairState := E_SlitPairStates.GEAROUT_BLADES;
        END_IF

    E_SlitPairStates.GEAROUT_BLADES: //Clear amy residual gearing
        actClearSlitGearing();
        eSlitPairState := E_SlitPairStates.CHECK_GEAROUT_COMPLETE;

    E_SlitPairStates.CHECK_GEAROUT_COMPLETE: //Check gearing cleared
        IF bBladesUncoupled THEN
            eSlitPairState := E_SlitPairStates.CLEAR_GAP_CALIBRATION; //Back to homing, this ensures the setpoint position of the axis is updated.
        END_IF

    E_SlitPairStates.CLEAR_GAP_CALIBRATION:
        mcHomeGapSize.Execute := TRUE;
        mcHomeGapCentre.Execute := TRUE;
        IF mcHomeGapSize.Done AND mcHomeGapCentre.Done THEN
            eSlitPairState := E_SlitPairStates.HOME_GAP; //Back to homing, this ensures the setpoint position of the axis is updated.
        END_IF

    E_SlitPairStates.ERROR: //ERROR STATE
        resetCounterTimeout := 0;
        bError := TRUE;
        bEnabled := FALSE;
        IF bReset THEN
            bResetting := TRUE;
            eSlitPairState := E_SlitPairStates.ERROR_GEAROUT;
        END_IF

    E_SlitPairStates.ERROR_GEAROUT: //Try to clear issues
        actClearSlitGearing();
        eSlitPairState := E_SlitPairStates.ERROR_GEAROUT_CHECK;

    E_SlitPairStates.ERROR_GEAROUT_CHECK:
        IF bBladesUncoupled THEN
            eSlitPairState := E_SlitPairStates.ERROR_RESET_AXES; //Back to homing, this ensures the setpoint position of the axis is updated.
        END_IF

    E_SlitPairStates.ERROR_RESET_AXES: //RESET ALL AXES
        GVL.astAxes[iBladeNegative].stControl.bReset := TRUE;
        GVL.astAxes[iBladePositive].stControl.bReset := TRUE;
        GVL.astAxes[iGapSize].stControl.bReset := TRUE;
        GVL.astAxes[iGapCentre].stControl.bReset := TRUE;
        resetCounterTimeout := resetCounterTimeout + 1;
        eSlitPairState := E_SlitPairStates.ERROR_RESET_CHECK;

    E_SlitPairStates.ERROR_RESET_CHECK:
        IF resetCounterTimeout > 10 THEN
            eSlitPairState := E_SlitPairStates.ERROR;
            bResetting := FALSE;
            RETURN;
        END_IF
        IF bAxisErrorsPresent THEN
            eSlitPairState := E_SlitPairStates.ERROR_RESET_AXES;
        ELSE
            eSlitPairState := E_SlitPairStates.INIT;
            bError := FALSE;
            bResetting := FALSE;
        END_IF
END_CASE
bReset := FALSE;

ACTION actClearSlitGearing:
//Action to send gearOut command to blade axes
GVL.astAxes[iBladeNegative].stControl.eCommand := E_MotionFunctions.eGearOut;
GVL.astAxes[iBladePositive].stControl.eCommand := E_MotionFunctions.eGearOut;
GVL.astAxes[iBladeNegative].stControl.bExecute := TRUE;
GVL.astAxes[iBladePositive].stControl.bExecute := TRUE;
END_ACTION

ACTION actErrorHandling:
//Error handling for slit functionality
IF bResetting THEN //ignore setting in error state if FB going through a reset
    RETURN;
END_IF

IF NOT bError AND bAxisErrorsPresent THEN
    eSlitPairState := E_SlitPairStates.ERROR;
END_IF
IF eSlitPairState <> E_SlitPairStates.INIT AND NOT bAxesEnabled THEN
    eSlitPairState := E_SlitPairStates.ERROR;
END_IF
IF (eSlitPairState <> E_SlitPairStates.INIT AND NOT bFunctionInErrorState) AND NOT bEnable THEN
    eSlitPairState := E_SlitPairStates.ERROR;
END_IF
IF bEnabled AND NOT bBladesHomed THEN
    eSlitPairState := E_SlitPairStates.ERROR;
END_IF
END_ACTION

ACTION actGapLimits:
//Set Virtual axis inputs to TRUE to enable movement
GVL.astAxes[iGapSize].stInputs.bLimitBwd := TRUE;
GVL.astAxes[iGapSize].stInputs.bLimitFwd := TRUE;
GVL.astAxes[iGapCentre].stInputs.bLimitBwd := TRUE;
GVL.astAxes[iGapCentre].stInputs.bLimitFwd := TRUE;
END_ACTION

ACTION actRunMethods:
checkAllAxesEnabled(bOutput => bAxesEnabled);
checkBladesHomed(bOutput => bBladesHomed);
checkVirtualHomed(bOutput => bGapHomed);
checkBladesCoupled(bOutput => bBladesCoupled);
checkBladesUncoupled(bOutput => bBladesUncoupled);
checkAllAxisErrors(bOutput => bAxisErrorsPresent);
checkErrorState(bOutput => bFunctionInErrorState);
END_ACTION

ACTION actSetupSlitGearing:
GVL.astAxes[iBladeNegative].stControl.eCommand := E_MotionFunctions.eGearInMultiMaster;
GVL.astAxes[iBladeNegative].stConfig.astMultiMasterAxis[1].nIndex := iGapSize;
GVL.astAxes[iBladeNegative].stConfig.astMultiMasterAxis[1].fRatio := -0.5;
GVL.astAxes[iBladeNegative].stConfig.astMultiMasterAxis[2].nIndex := iGapCentre;
GVL.astAxes[iBladeNegative].stConfig.astMultiMasterAxis[2].fRatio := 1;
GVL.astAxes[iBladePositive].stControl.eCommand := E_MotionFunctions.eGearInMultiMaster;
GVL.astAxes[iBladePositive].stConfig.astMultiMasterAxis[1].nIndex := iGapSize;
GVL.astAxes[iBladePositive].stConfig.astMultiMasterAxis[1].fRatio := 0.5;
GVL.astAxes[iBladePositive].stConfig.astMultiMasterAxis[2].nIndex := iGapCentre;
GVL.astAxes[iBladePositive].stConfig.astMultiMasterAxis[2].fRatio := 1;
GVL.astAxes[iBladeNegative].stControl.bExecute := TRUE;
GVL.astAxes[iBladePositive].stControl.bExecute := TRUE;
END_ACTION

ACTION actVirtualAxisPositions:
(*Calculate virtual axis positions and convert to UDINT.
Conversion to UDINT is prohibited if it would exceed UDINT max value of 4,294,967,295.
If this is not done, it can cause overflow when connected to the encoder input and hard-crash the PLC which will only recover with a power cycle.
To preserve decimal position data of the LREAL (i.e. anything <1mm) it is necessary to scale the value before converting to UDINT.
This can be reversed with the correct scaling at the NC encoder level.
*)
fGapSizePosition := GVL.astAxes[iBladePositive].stStatus.fActPosition - GVL.astAxes[iBladeNegative].stStatus.fActPosition;
fGapCentrePosition := (GVL.astAxes[iBladePositive].stStatus.fActPosition + GVL.astAxes[iBladeNegative].stStatus.fActPosition) / 2;

IF bBladesHomed THEN
    IF ABS(fGapSizePosition) < 100000 THEN
        iGapSizePosition := LREAL_TO_UDINT(fGapSizePosition*fEncoderScaling);
    END_IF
    IF ABS(fGapCentrePosition) < 100000 THEN
        iGapCentrePosition := LREAL_TO_UDINT(fGapCentrePosition*fEncoderScaling);
    END_IF
END_IF
END_ACTION

(*Method to check if all axes (real and virtual) are enabled.
Only returns TRUE if BOTH blades are homed*)
METHOD checkAllAxesEnabled: BOOL
VAR_OUTPUT
    bOutput: BOOL:= TRUE;
END_VAR
IF NOT GVL.astAxes[iBladeNegative].stStatus.bEnabled THEN
    bOutput := FALSE;
END_IF
IF NOT GVL.astAxes[iBladePositive].stStatus.bEnabled THEN
    bOutput := FALSE;
END_IF
IF NOT GVL.astAxes[iGapSize].stStatus.bEnabled THEN
    bOutput := FALSE;
END_IF
IF NOT GVL.astAxes[iGapCentre].stStatus.bEnabled THEN
    bOutput := FALSE;
END_IF
END_METHOD

(*Method to check if an error is present on any axis.
Returns TRUE if an error is present on any axis *)
METHOD checkAllAxisErrors: BOOL
VAR_OUTPUT
    bOutput: BOOL := FALSE;
END_VAR
IF GVL.astAxes[iGapSize].stStatus.bError THEN
    bOutput := TRUE;
END_IF
IF GVL.astAxes[iGapCentre].stStatus.bError THEN
    bOutput := TRUE;
END_IF
IF GVL.astAxes[iBladeNegative].stStatus.bError THEN
    bOutput := TRUE;
END_IF
IF GVL.astAxes[iBladePositive].stStatus.bError THEN
    bOutput := TRUE;
END_IF
END_METHOD

(*Method to check if both blades are coupled to the virtual axes.
Only returns TRUE if BOTH blades are coupled *)
METHOD checkBladesCoupled: BOOL
VAR_OUTPUT
    bOutput: BOOL := TRUE;
END_VAR
IF NOT GVL.astAxes[iBladeNegative].stStatus.bGeared THEN
    bOutput := FALSE;
END_IF
IF NOT GVL.astAxes[iBladePositive].stStatus.bGeared THEN
    bOutput := FALSE;
END_IF
END_METHOD

(*Method to check if blade axes are homed/have the calibration flag.
Only returns TRUE if BOTH blades are homed*)
METHOD checkBladesHomed: BOOL
VAR_OUTPUT
    bOutput: BOOL := TRUE;
END_VAR
IF NOT GVL.astAxes[iBladeNegative].stStatus.bHomed THEN
    bOutput := FALSE;
END_IF
IF NOT GVL.astAxes[iBladePositive].stStatus.bHomed THEN
    bOutput := FALSE;
END_IF
END_METHOD

(*Method to check if both blades are uncoupled from the virtual axes.
Only returns TRUE if BOTH blades are uncoupled *)
METHOD checkBladesUncoupled: BOOL
VAR_OUTPUT
    bOutput: BOOL:= TRUE;
END_VAR
IF GVL.astAxes[iBladeNegative].stStatus.bGeared THEN
    bOutput := FALSE;
END_IF
IF GVL.astAxes[iBladePositive].stStatus.bGeared THEN
    bOutput := FALSE;
END_IF
END_METHOD

METHOD checkErrorState: BOOL
VAR_OUTPUT
    bOutput: BOOL := FALSE;
END_VAR
IF eSlitPairState = E_SlitPairStates.ERROR THEN
    bOutput := TRUE;
END_IF
IF eSlitPairState = E_SlitPairStates.ERROR_GEAROUT THEN
    bOutput := TRUE;
END_IF
IF eSlitPairState = E_SlitPairStates.ERROR_GEAROUT_CHECK THEN
    bOutput := TRUE;
END_IF
IF eSlitPairState = E_SlitPairStates.ERROR_RESET_AXES THEN
    bOutput := TRUE;
END_IF
IF eSlitPairState = E_SlitPairStates.ERROR_RESET_CHECK THEN
    bOutput := TRUE;
END_IF
END_METHOD

(*Method to check if the virtual axes for gap size and gap centre are homed/the calibration flag is present.
Only returns TRUE if BOTH virtual axes are homed *)
METHOD checkVirtualHomed: BOOL
VAR_OUTPUT
    bOutput: BOOL:= TRUE;
END_VAR
IF NOT GVL.astAxes[iGapSize].stStatus.bHomed THEN
    bOutput := FALSE;
END_IF
IF NOT GVL.astAxes[iGapCentre].stStatus.bHomed THEN
    bOutput := FALSE;
END_IF
END_METHOD

END_FUNCTION_BLOCK

// ---- tc_mca_std_lib/POUs/Motion/FB_SlitPairV2.TcPOU

FUNCTION_BLOCK FB_SlitPairV2
VAR_INPUT
    nIdPositiveAxis: UINT; //ID of axis for which positive motion increases gap size
    nIdNegativeAxis: UINT; //ID of axis for which negative motion increases gap size
    nIdGapSizeAxis: UINT; //ID of virtual gap aperture size axis
    nIdGapCentreAxis: UINT; //ID of virtual gap centre position axis

    bEnable: BOOL; //Enable slit pair logic functionality
    bReset: BOOL; //Reset from error state
    fEncoderScaling: LREAL := 10000; //Virtual axis scaling denominator, default of 10000
END_VAR
VAR
    nGapSizeEncoder AT %Q*: UDINT := 0;
    nGapCentreEncoder AT %Q*: UDINT := 0;
    fGapSize: LREAL;
    fGapCentre: LREAL;
    bAllHalted: BOOL := FALSE;
    bInternalResetHome: BOOL :=FALSE;

    fbSetpointGenEnablePositiveAxis: MC_ExtSetPointGenEnable;
    fbSetpointGenEnableNegativeAxis: MC_ExtSetPointGenEnable;
    fbSetpointGenEnableGapSizeAxis: MC_ExtSetPointGenEnable;
    fbSetpointGenEnableGapCentreAxis: MC_ExtSetPointGenEnable;

    fbSetpointGenDisablePositiveAxis: MC_ExtSetPointGenDisable;
    fbSetpointGenDisableNegativeAxis: MC_ExtSetPointGenDisable;
    fbSetpointGenDisableGapSizeAxis: MC_ExtSetPointGenDisable;
    fbSetpointGenDisableGapCentreAxis: MC_ExtSetPointGenDisable;

    fPosSetpointPositiveAxis: LREAL;
    fPosSetpointNegativeAxis: LREAL;
    fPosSetpointGapSizeAxis: LREAL;
    fPosSetpointGapCentreAxis: LREAL;

    fVeloSetpointPositiveAxis: LREAL;
    fVeloSetpointNegativeAxis: LREAL;
    fVeloSetpointGapSizeAxis: LREAL;
    fVeloSetpointGapCentreAxis: LREAL;

    nDirectionPositiveAxis: DINT;
    nDirectionNegativeAxis: DINT;
    nDirectionGapSizeAxis: DINT;
    nDirectionGapCentreAxis: DINT;

    eState: E_SlitPairStatesV2 := E_SlitPairStatesV2.eInit;

    bInternalReset: BOOL;
    bHomingReset: BOOL := FALSE;

    //Two resets required due to homing functionality
    bResetInProgressCheck1: BOOL := FALSE;
    bResetInProgressCheck2: BOOL := FALSE;

    //internal MCPOWER blocks because Beckhoff won't let you enable a setpoint generator on a limit....
    fbPowerPositiveAxis: MC_POWER;
    fbPowerNegativeAxis: MC_POWER;
    fbPowerGapSizeAxis: MC_POWER;
    fbPowerGapCentreAxis: MC_POWER;

    //internal MC_Reset, needed because the current reset in FB_Axis works only when there is an error. This should change once the reset functionality changes
    fbInternalResetTrig: R_TRIG;
    fbInternalResetHome: R_TRIG;
    fbResetPositiveAxis: MC_RESET;
    fbResetNegativeAxis: MC_RESET;
    fbResetGapSizeAxis: MC_RESET;
    fbResetGapCentreAxis: MC_RESET;
    fbResetHomedGap: MC_Home;
    fbResetHomedCentre: MC_Home;

END_VAR


(*SETUP INSTRUCTIONS
Virtual axes:
Encoder type set to Universal
Encoder mask set to 0xFFFFFFFF
Encoder scaling set to match FB
Link nDataIn1 of encoder to FB encoders
Position lag monitoring can be left on*
Dynamics of virtual axes must be configured considering coupled mechanicals (e.g. don't set velocities your real axes can't achieve)
*)

//Position of virtual axes
actVirtualAxisPositions();
//Limit logic
actVirtualAxisLimits();
//Enable Logic - Virtual axes automatically enable when real axes are enabled
actVirtualAxisEnable();
//Call spGenerator FBs
actGeneratorEnableDisable();
//Calculate position setpoints
actCalculateSetpointPositions();
//Calculate velocity setpoints
actCalculateSetpointVelocities();
//Calculate directions
actCalculateSetpointDirections();

//Error state handling - only handle errors that disable motion
IF bEnable AND (GVL.astAxes[nIdPositiveAxis].Axis.Status.ErrorStop OR GVL.astAxes[nIdNegativeAxis].Axis.Status.ErrorStop OR GVL.astAxes[nIdGapSizeAxis].Axis.Status.ErrorStop OR GVL.astAxes[nIdGapCentreAxis].Axis.Status.ErrorStop) THEN
    eState := E_SlitPairStatesV2.eError;
END_IF

//Propagate real axis error to virtual
IF GVL.astAxes[nIdPositiveAxis].Axis.Status.ErrorStop AND (NOT GVL.astAxes[nIdGapSizeAxis].Axis.Status.ErrorStop OR NOT GVL.astAxes[nIdGapCentreAxis].Axis.Status.ErrorStop) THEN
    GVL.astAxes[nIdGapSizeAxis].stStatus.bError := TRUE;
    GVL.astAxes[nIdGapCentreAxis].stStatus.bError := TRUE;
    GVL.astAxes[nIdGapSizeAxis].stStatus.nErrorID := GVL.astAxes[nIdPositiveAxis].stStatus.nErrorID;
    GVL.astAxes[nIdGapCentreAxis].stStatus.nErrorID := GVL.astAxes[nIdPositiveAxis].stStatus.nErrorID;
ELSIF  GVL.astAxes[nIdNegativeAxis].Axis.Status.ErrorStop AND (NOT GVL.astAxes[nIdGapSizeAxis].Axis.Status.ErrorStop OR NOT GVL.astAxes[nIdGapCentreAxis].Axis.Status.ErrorStop) THEN
    GVL.astAxes[nIdGapSizeAxis].stStatus.bError := TRUE;
    GVL.astAxes[nIdGapCentreAxis].stStatus.bError := TRUE;
    GVL.astAxes[nIdGapSizeAxis].stStatus.nErrorID := GVL.astAxes[nIdNegativeAxis].stStatus.nErrorID;
    GVL.astAxes[nIdGapCentreAxis].stStatus.nErrorID := GVL.astAxes[nIdNegativeAxis].stStatus.nErrorID;
END_IF

//Internal Reset linked to any axis reset
bInternalReset := bReset OR GVL.astAxes[nIdPositiveAxis].stControl.bReset OR GVL.astAxes[nIdNegativeAxis].stControl.bReset OR GVL.astAxes[nIdGapSizeAxis].stControl.bReset OR GVL.astAxes[nIdGapCentreAxis].stControl.bReset;

//If real axis is homing, change state
IF bEnable AND (GVL.astAxes[nIdPositiveAxis].Axis.Status.HomingBusy OR GVL.astAxes[nIdNegativeAxis].Axis.Status.HomingBusy) THEN
    eState := E_SlitPairStatesV2.eWaitForRealHomed;
END_IF

//Link all halt buttons in motors
IF GVL.astAxes[nIdPositiveAxis].stControl.bHalt OR GVL.astAxes[nIdNegativeAxis].stControl.bHalt OR
    GVL.astAxes[nIdGapSizeAxis].stControl.bHalt OR GVL.astAxes[nIdGapCentreAxis].stControl.bHalt THEN
    actHaltAllAxes();
END_IF

//Propagate homing status
fbResetHomedGap(Axis:= GVL.astAxes[nIdGapSizeAxis].Axis, HomingMode:= MC_ResetCalibration);
fbResetHomedCentre(Axis:= GVL.astAxes[nIdGapCentreAxis].Axis, HomingMode:= MC_ResetCalibration);
fbInternalResetHome(CLK:= fbResetHomedCentre.Done OR fbResetHomedGap.Done );
IF NOT GVL.astAxes[nIdPositiveAxis].stStatus.bHomed OR NOT GVL.astAxes[nIdNegativeAxis].stStatus.bHomed THEN
        fbResetHomedGap.Execute := TRUE;
        fbResetHomedCentre.Execute := TRUE;
END_IF

IF fbInternalResetHome.Q THEN
        fbResetHomedGap.Execute := FALSE;
        fbResetHomedCentre.Execute := FALSE;
END_IF


//State machine
IF bEnable THEN
    CASE eState OF  //HOMING LOOP ISSUE
        E_SlitPairStatesV2.eInit:
            //If real axes are calibrated, then home the virtual axes, else go Operatioanl
            fbResetPositiveAxis(Axis:=GVL.astAxes[nIdPositiveAxis].Axis, Execute:=FALSE);
            fbResetNegativeAxis(Axis:=GVL.astAxes[nIdNegativeAxis].Axis, Execute:=FALSE);
            fbResetGapSizeAxis(Axis:=GVL.astAxes[nIdGapSizeAxis].Axis, Execute:=FALSE);
            fbResetGapCentreAxis(Axis:=GVL.astAxes[nIdGapCentreAxis].Axis, Execute:=FALSE);
            IF GVL.astAxes[nIdPositiveAxis].stStatus.bHomed AND GVL.astAxes[nIdNegativeAxis].stStatus.bHomed THEN
               GVL.astAxes[nIdGapSizeAxis].stConfig.eHomeSeq := E_HomingRoutines.eHomeDirect;
               GVL.astAxes[nIdGapCentreAxis].stConfig.eHomeSeq := E_HomingRoutines.eHomeDirect;
               GVL.astAxes[nIdGapSizeAxis].stConfig.fHomePosition := fGapSize;
               GVL.astAxes[nIdGapCentreAxis].stConfig.fHomePosition := fGapCentre;
                eState := E_SlitPairStatesV2.eWaitForVirtualHomed;
            ELSE
                eState := E_SlitPairStatesV2.eOperational;
            END_IF

        E_SlitPairStatesV2.eWaitForVirtualHomed:
            //Wait for virtual axis homing to complete/
            GVL.astAxes[nIdGapSizeAxis].stControl.eCommand := E_MotionFunctions.eHome;
            GVL.astAxes[nIdGapSizeAxis].stControl.bExecute := TRUE;
            GVL.astAxes[nIdGapCentreAxis].stControl.eCommand := E_MotionFunctions.eHome;
            GVL.astAxes[nIdGapCentreAxis].stControl.bExecute := TRUE;
            IF GVL.astAxes[nIdGapSizeAxis].stStatus.bHomed AND GVL.astAxes[nIdGapCentreAxis].stStatus.bHomed THEN
                eState := E_SlitPairStatesV2.eOperational;
            END_IF
            //IF NOT IN HOMING STATE

        E_SlitPairStatesV2.eOperational:
            bResetInProgressCheck1 := FALSE;
            //Detect whether real or virtual axes are moving
            IF GVL.astAxes[nIdGapSizeAxis].stStatus.bMoving OR GVL.astAxes[nIdGapCentreAxis].stStatus.bMoving THEN
                eState := E_SlitPairStatesV2.eEnableRealGenerators;
            END_IF
            IF GVL.astAxes[nIdPositiveAxis].stStatus.bMoving OR GVL.astAxes[nIdNegativeAxis].stStatus.bMoving THEN
                eState := E_SlitPairStatesV2.eEnableVirtualGenerators;
            END_IF

        E_SlitPairStatesV2.eEnableRealGenerators:
            //Hold MC_Power on until generators have enabled
            fbPowerPositiveAxis(Axis:=GVL.astAxes[nIdPositiveAxis].Axis, Enable:=TRUE, Enable_Positive:=TRUE,Enable_Negative:=TRUE);
            fbPowerNegativeAxis(Axis:=GVL.astAxes[nIdNegativeAxis].Axis, Enable:=TRUE, Enable_Positive:=TRUE,Enable_Negative:=TRUE);
            fbSetpointGenEnablePositiveAxis.Execute := TRUE;
            fbSetpointGenEnableNegativeAxis.Execute := TRUE;
            eState := E_SlitPairStatesV2.eCheckRealAxisGeneratorsEnabled;

        E_SlitPairStatesV2.eCheckRealAxisGeneratorsEnabled:
            //Hold MC_Power on until generators have enabled
            fbPowerPositiveAxis(Axis:=GVL.astAxes[nIdPositiveAxis].Axis, Enable:=TRUE, Enable_Positive:=TRUE,Enable_Negative:=TRUE);
            fbPowerNegativeAxis(Axis:=GVL.astAxes[nIdNegativeAxis].Axis, Enable:=TRUE, Enable_Positive:=TRUE,Enable_Negative:=TRUE);
            IF fbSetpointGenEnablePositiveAxis.Enabled AND fbSetpointGenEnableNegativeAxis.Enabled THEN
                eState := E_SlitPairStatesV2.eWaitForVirtualMoveDone;
            END_IF

        E_SlitPairStatesV2.eWaitForVirtualMoveDone:
            IF NOT(GVL.astAxes[nIdGapSizeAxis].stStatus.bMoving OR GVL.astAxes[nIdGapCentreAxis].stStatus.bMoving) THEN
                eState := E_SlitPairStatesV2.eDisableRealGenerators;
            END_IF

        E_SlitPairStatesV2.eDisableRealGenerators:
            fbSetpointGenDisablePositiveAxis.Execute := TRUE;
            fbSetpointGenDisableNegativeAxis.Execute := TRUE;
            eState := E_SlitPairStatesV2.eOperational;

        E_SlitPairStatesV2.eEnableVirtualGenerators:
            //Hold MC_Power on until generators have enabled
            fbPowerGapSizeAxis(Axis:=GVL.astAxes[nIdGapSizeAxis].Axis, Enable:=TRUE, Enable_Positive:=TRUE,Enable_Negative:=TRUE);
            fbPowerGapCentreAxis(Axis:=GVL.astAxes[nIdGapCentreAxis].Axis, Enable:=TRUE, Enable_Positive:=TRUE,Enable_Negative:=TRUE);
            fbSetpointGenEnableGapSizeAxis.Execute := TRUE;
            fbSetpointGenEnableGapCentreAxis.Execute := TRUE;
            eState := E_SlitPairStatesV2.eCheckVirtualAxisGeneratorsEnabled;

        E_SlitPairStatesV2.eCheckVirtualAxisGeneratorsEnabled:
            //Hold MC_Power on until generators have enabled
            fbPowerGapSizeAxis(Axis:=GVL.astAxes[nIdGapSizeAxis].Axis, Enable:=TRUE, Enable_Positive:=TRUE,Enable_Negative:=TRUE);
            fbPowerGapCentreAxis(Axis:=GVL.astAxes[nIdGapCentreAxis].Axis, Enable:=TRUE, Enable_Positive:=TRUE,Enable_Negative:=TRUE);
            IF fbSetpointGenEnableGapSizeAxis.Enabled AND fbSetpointGenEnableGapCentreAxis.Enabled THEN
                eState := E_SlitPairStatesV2.eWaitForRealMoveDone;
            END_IF

        E_SlitPairStatesV2.eWaitForRealMoveDone:
            IF NOT(GVL.astAxes[nIdPositiveAxis].stStatus.bMoving OR GVL.astAxes[nIdNegativeAxis].stStatus.bMoving) THEN
                eState := E_SlitPairStatesV2.eDisableVirtualGenerators;
            END_IF

        E_SlitPairStatesV2.eDisableVirtualGenerators:
            fbSetpointGenDisableGapSizeAxis.Execute := TRUE;
            fbSetpointGenDisableGapCentreAxis.Execute := TRUE;
            eState := E_SlitPairStatesV2.eOperational;

        E_SlitPairStatesV2.eError:
            actHaltAllAxes();

            IF bHomingReset THEN
                bInternalReset := TRUE;
                bResetInProgressCheck1 := TRUE;
                bResetInProgressCheck2 := TRUE;
                bHomingReset := FALSE;
            END_IF
            IF bInternalReset OR bReset OR bResetInProgressCheck2 THEN
                fbResetPositiveAxis(Axis:=GVL.astAxes[nIdPositiveAxis].Axis, Execute:=TRUE);
                fbResetNegativeAxis(Axis:=GVL.astAxes[nIdNegativeAxis].Axis, Execute:=TRUE);
                fbResetGapSizeAxis(Axis:=GVL.astAxes[nIdGapSizeAxis].Axis, Execute:=TRUE);
                fbResetGapCentreAxis(Axis:=GVL.astAxes[nIdGapCentreAxis].Axis, Execute:=TRUE);
                GVL.astAxes[nIdPositiveAxis].stControl.bReset := TRUE;
                GVL.astAxes[nIdNegativeAxis].stControl.bReset := TRUE;
                GVL.astAxes[nIdGapSizeAxis].stControl.bReset := TRUE;
                GVL.astAxes[nIdGapCentreAxis].stControl.bReset := TRUE;
                IF NOT(bResetInProgressCheck1) THEN
                    bResetInProgressCheck2 := FALSE;
                END_IF
            END_IF

            IF NOT(GVL.astAxes[nIdPositiveAxis].stStatus.bError) AND NOT(GVL.astAxes[nIdNegativeAxis].stStatus.bError) AND NOT(GVL.astAxes[nIdGapSizeAxis].stStatus.bError) AND NOT(GVL.astAxes[nIdGapCentreAxis].stStatus.bError) THEN
                eState := E_SlitPairStatesV2.eInit;
            END_IF

        E_SlitPairStatesV2.eWaitForRealHomed:
            bHomingReset := TRUE;
            IF NOT GVL.astAxes[nIdPositiveAxis].Axis.Status.Homed OR NOT GVL.astAxes[nIdNegativeAxis].Axis.Status.Homed THEN
                eState := E_SlitPairStatesV2.eInit;
            END_IF
    END_CASE
END_IF


//Feed externalsetpoint generators setpoint values - ignoring acceleration
MC_ExtSetPointGenFeed(Axis:= GVL.astAxes[nIdPositiveAxis].Axis, Position:= fPosSetpointPositiveAxis, Velocity:= fVeloSetpointPositiveAxis, Acceleration:= 0, Direction:= nDirectionPositiveAxis);
MC_ExtSetPointGenFeed(Axis:= GVL.astAxes[nIdNegativeAxis].Axis, Position:= fPosSetpointNegativeAxis, Velocity:= fVeloSetpointNegativeAxis, Acceleration:= 0, Direction:= nDirectionNegativeAxis);
MC_ExtSetPointGenFeed(Axis:= GVL.astAxes[nIdGapSizeAxis].Axis, Position:= fPosSetpointGapSizeAxis, Velocity:= fVeloSetpointGapSizeAxis, Acceleration:= 0, Direction:= nDirectionGapSizeAxis);
MC_ExtSetPointGenFeed(Axis:= GVL.astAxes[nIdGapCentreAxis].Axis, Position:= fPosSetpointGapCentreAxis, Velocity:= fVeloSetpointGapCentreAxis, Acceleration:= 0, Direction:= nDirectionGapCentreAxis);

bReset := FALSE;

ACTION actCalculateSetpointDirections:

IF fVeloSetpointPositiveAxis > 0 THEN
    nDirectionPositiveAxis := 1; //moving forward
ELSIF fVeloSetpointPositiveAxis < 0 THEN
    nDirectionPositiveAxis := -1; //moving backward
ELSE
    nDirectionPositiveAxis := 0; //stationary
END_IF

IF fVeloSetpointNegativeAxis > 0 THEN
    nDirectionNegativeAxis := 1; //moving forward
ELSIF fVeloSetpointNegativeAxis < 0 THEN
    nDirectionNegativeAxis := -1; //moving backward
ELSE
    nDirectionNegativeAxis := 0; //stationary
END_IF

IF fVeloSetpointGapSizeAxis > 0 THEN
    nDirectionGapSizeAxis := 1; //moving forward
ELSIF fVeloSetpointGapSizeAxis < 0 THEN
    nDirectionGapSizeAxis := -1; //moving backward
ELSE
    nDirectionGapSizeAxis := 0; //stationary
END_IF

IF fVeloSetpointGapCentreAxis > 0 THEN
    nDirectionGapCentreAxis := 1; //moving forward
ELSIF fVeloSetpointGapCentreAxis < 0 THEN
    nDirectionGapCentreAxis := -1; //moving backward
ELSE
    nDirectionGapCentreAxis := 0; //stationary
END_IF
END_ACTION

ACTION actCalculateSetpointPositions:

fPosSetpointPositiveAxis := GVL.astAxes[nIdGapCentreAxis].Axis.NcToPlc.SetPos + (GVL.astAxes[nIdGapSizeAxis].Axis.NcToPlc.SetPos/2);
fPosSetpointNegativeAxis := GVL.astAxes[nIdGapCentreAxis].Axis.NcToPlc.SetPos - (GVL.astAxes[nIdGapSizeAxis].Axis.NcToPlc.SetPos/2);
fPosSetpointGapSizeAxis := GVL.astAxes[nIdPositiveAxis].Axis.NcToPlc.SetPos - GVL.astAxes[nIdNegativeAxis].Axis.NcToPlc.SetPos;
fPosSetpointGapCentreAxis := (GVL.astAxes[nIdPositiveAxis].Axis.NcToPlc.SetPos + GVL.astAxes[nIdNegativeAxis].Axis.NcToPlc.SetPos) / 2;
END_ACTION

ACTION actCalculateSetpointVelocities:

fVeloSetpointPositiveAxis := GVL.astAxes[nIdGapCentreAxis].Axis.NcToPlc.SetVelo +(GVL.astAxes[nIdGapSizeAxis].Axis.NcToPlc.SetVelo/2);
fVeloSetpointNegativeAxis := GVL.astAxes[nIdGapCentreAxis].Axis.NcToPlc.SetVelo -(GVL.astAxes[nIdGapSizeAxis].Axis.NcToPlc.SetVelo/2);
fVeloSetpointGapSizeAxis := GVL.astAxes[nIdPositiveAxis].Axis.NcToPlc.SetVelo - GVL.astAxes[nIdNegativeAxis].Axis.NcToPlc.SetVelo;
fVeloSetpointGapCentreAxis := GVL.astAxes[nIdPositiveAxis].Axis.NcToPlc.SetVelo + GVL.astAxes[nIdNegativeAxis].Axis.NcToPlc.SetVelo;
END_ACTION

ACTION actGeneratorEnableDisable:

fbSetpointGenEnablePositiveAxis(Axis:=GVL.astAxes[nIdPositiveAxis].Axis);
fbSetpointGenEnablePositiveAxis.Execute := FALSE;

fbSetpointGenEnableNegativeAxis(Axis:=GVL.astAxes[nIdNegativeAxis].Axis);
fbSetpointGenEnableNegativeAxis.Execute := FALSE;

fbSetpointGenEnableGapSizeAxis(Axis:=GVL.astAxes[nIdGapSizeAxis].Axis);
fbSetpointGenEnableGapSizeAxis.Execute := FALSE;

fbSetpointGenEnableGapCentreAxis(Axis:=GVL.astAxes[nIdGapCentreAxis].Axis);
fbSetpointGenEnableGapCentreAxis.Execute := FALSE;


fbSetpointGenDisablePositiveAxis(Axis:=GVL.astAxes[nIdPositiveAxis].Axis);
fbSetpointGenDisablePositiveAxis.Execute := FALSE;

fbSetpointGenDisableNegativeAxis(Axis:=GVL.astAxes[nIdNegativeAxis].Axis);
fbSetpointGenDisableNegativeAxis.Execute := FALSE;

